	fbLys		: FB_Light_Type_A;
	
	stDaliSetup	: SH_Light.ST_DALI_RoomSetup := (		byShrtAdr_Prim := 10, 
														byGrpAdr_Prim := 2, 
														eMod_Prim := E_DALIAddressType.Group, 
													//	byShrtAdr_Sec := 1, 
													//	byGrpAdr_Sec := 1, 
													//	eMod_Sec := E_DALIAddressType.Short, 
													//	byShrtAdr_Supl := 1, 
														DALI_LINE_NUM_PRIM := 3, 
														DALI_LINE_NUM_SEC := 0, 
														DALI_LINE_NUM_SUPL := 0);
	stLiveData				: SH_Light.ST_LiveData;
	//stLiveData AT %MB22	: SH_Light.ST_LiveData;
	bTopButtonZone1			: BOOL;
	bTopButtonZone1_Visu	: BOOL;
	bBottomButtonZone1		: BOOL;
	bBottomButtonZone1_Visu	: BOOL;
	bButtonZone2			: BOOL;
	fLuxOn					: REAL;
	fLuxDim					: REAL;
	tPIRDim					: TIME;
	tPIROff					: TIME;
	fOffsetSec				: REAL := 20;
	bOccupiedRoom			: BOOL;

	bRunTuning				: BOOL;
	
// Sensor Settings
	//fbSensor					: SH_Light.FB_NIKO_P46xx_1Pcs;
	fbSensor					: SH_Light.FB_NIKO_P46xx_2Pcs;
	//bySensorAddr				: BYTE := 3;
	arrSensorAddr				: ARRAY[1..2] OF BYTE := [1,2];
	bInitialize					: BOOL := TRUE;
	stDaliSensorSetup			: ST_DALI_NIKOP46SetupData := (
																nSensitivityPIRSegmentA := arrSensitivityOccupancy[1],
																nSensitivityPIRSegmentB := arrSensitivityOccupancy[2],
																nSensitivityPIRSegmentC := arrSensitivityOccupancy[3]);
//	arrSensitivityOccupancy				: ARRAY[1..3] OF BYTE := [4,4,4];

	//bInitErr					: BOOL;
	//bInitDone					: BOOL;
	arrInitErr					: ARRAY [1..2] OF BOOL;
	arrInitDone					: ARRAY [1..2] OF BOOL;
	arrSensorScales				: ARRAY [1..10] OF SH_Light.ST_DALI_SensorScaleMode := [	(fMeassureMaxSensor := rMeassure_Zone5, fReadMaxSensor := rRead_Zone5),
																							(fMeassureMaxSensor := rMeassure_Zone5, fReadMaxSensor := rRead_Zone5),
																						8(())];
	bCancelHoldTimerOccupancy	: BOOL;
(*	eEventPriorityOccupancy		: E_DALIEventPriority := E_DALIEVENTPRIORITY.Middle;
	nHoldTimerOccupancy			: WORD := 5; // Value in s. 	
	nReportTimerOccupancy		: BYTE := 120; // Value in s, Preset manufacturer value
	nDeadtimeTimerOccupancy		: WORD := 100; // Value in ms, Predefined Value of DALI Standard
	bCancelHoldTimerOccupancy	: BOOL;
	nSensitivityOccupancy		: BYTE:= 3; //setting Sensivity (0..4) 0 (Off), 1 (Min), 2(Low), 3(High) and 4 (Max)

	bEnableLuxEvent				: BOOL;
	eEventPriorityBrightness	: E_DALIEventPriority := E_DALIEVENTPRIORITY.Middle;
	nDeadtimeTimerBrightness	: WORD := 1500; // Value in ms, Predefined Value of DALI Standard
	nHysteresisBrightness		: BYTE := 2; // Value in %
	nHysteresisMinBrightness	: BYTE := 10; // Absolute Value, depending on the manufacturer specific resolution
	nReportTimerBrightness		: BYTE := 120; // Value in s, Preset manufacturer value
*)



//ModbusComm setup
	
	fbWriteSPLuxLevel			: SH_Light.FB_TwoVal_SelectOne_RTrigChange;
	fbWritePirDelayTIme			: SH_Light.FB_TwoVal_SelectOne_RTrigChange;
	stRoomDataPLC				: SH_Light.ST_RoomDataPLC	:=	(	uiPirOffDelayTime	:= 30,
																	uiSpLuxLevel		:= 500,
																	uiPirDimDelayTime	:= 15,
																	uiSpDimLuxLevel		:= 200
																);
	fbBallastOnHours			: SH_Light.FB_CountOnHours;
	bEnableHourCount			: BOOL := TRUE;
	
	//Non-persistent modbus data
	bPirActive_MB			AT%MX32.0	: BOOL;				//bPirLys i gammel kode
	uiActLuxLevel_MB		AT%MB36	: UINT;				//intHMIAktueltLux i gammel kode
	uiActLightLevelPct_MB	AT%MB42		: UINT;				//intDALI_Gruppe1_Lysniveau i gammel kode
	
	//For Conversion
	uiPirOffMinutes						: UINT;
	udTimeScaling						: UDINT := 60000;
	uiLuxOn								: UINT;
	
	//max values checks
	uiMaxLuxLevel						: UINT := 1023;
	uiMaxPirOffMinutes					: UINT := 180;
	
END_VAR

VAR CONSTANT
Sensor_DALI_LINE_NUM: BYTE := 4;
	DALI_LINE_NUM_LIGHT: BYTE := 3;
	arrSensitivityOccupancy				: ARRAY[1..3] OF BYTE := [4,4,4];
END_VAR
VAR PERSISTENT
	stPirSensorData: SH_Light.ST_DALI_Sensor;
	stTuneData: SH_Light.ST_TuneData_EX;
	
	uiPirOffDelayTime_MB	AT%MB34		: UINT;				//ntHMI_Pir_SetValue i gammel kode
	uiSPLuxLevel_MB			AT%MB38 	: UINT;				//intHMI_Lux_SetValue i gammel kode
	uiBallastOnHours_MB		AT%MB46 	: UINT;				//dintHMILysbraendtimer1 i gammel kode
	byOnHoursOverflowCount				: BYTE;
END_VAR

A_Buttons();
A_LightCtrl();
A_Sensor();
A_Modbuscomm();

ACTION A_Buttons:
bTopButtonZone1		:= GVL_EnOcean.strEnOceanSwitch_Rum_3_329_Indgang.bT1_ON OR GVL_EnOcean.strEnOceanSwitch_Rum_3_329_Tavle.bT2_OFF OR bTopButtonZone1_Visu;
bBottomButtonZone1	:= GVL_EnOcean.strEnOceanSwitch_Rum_3_329_Indgang.bT1_OFF OR GVL_EnOcean.strEnOceanSwitch_Rum_3_329_Tavle.bT2_ON OR bBottomButtonZone1_Visu;
END_ACTION

ACTION A_LightCtrl:

fbLys(
	nZoneID:= 1, 
	bButtonZone1:= bTopButtonZone1,
	bBottomButtonZone1 := bBottomButtonZone1, 
	bButtonZone2:= bButtonZone2, 
	fLuxOn:= fLuxOn, 
	fLuxDim:= fLuxDim, 
	tPIRDim:= tPIRDim, 
	tPIROff:= tPIROff, 
	fOffsetSec:= fOffsetSec, 
	bReInit:= , 
	stDaliSetup:= stDaliSetup, 
	ipCommunication_Prim:= P_DALI_Background.arrfbKL6821Communication[DALI_LINE_NUM_LIGHT], 
//	ipCommunication_Sec:= P_DALI_Background.arrfbKL6821Communication[DALI_LINE_NUM_LIGHT], 
//	ipCommunication_Supl:= P_DALI_Background.arrfbKL6821Communication[DALI_LINE_NUM_LIGHT], 
	fMinOutputPowerLevelRoom:= 15, 
	fMaxOutputPowerLevelRoom:= 100, 
	nCycleTimeInMS:= SH_Light.DALI_Param.nPlcTaskCycleTimeInMS*nDimCmdCycleTimeFactor, 
	bRunTuning:= bRunTuning, 
	bOccupiedRoom=> bOccupiedRoom, 
	bError_Prim=> , 
	nError_Prim=> , 
	stTuneData:=stTuneData , 
	stPirSensorData:= stPirSensorData, 
	stLiveData:= stLiveData);
END_ACTION

ACTION A_ModbusComm:
//Manage data for modbus communication

//Manage data for read-only in PLC
stRoomDataPLC.bPirActive			:= stPirSensorData.bPrc;
stRoomDataPLC.uiActLuxLevel			:= TO_UINT(TRUNC(stPirSensorData.fBrightness));
stRoomDataPLC.uiActLightLevelPct	:= TO_UINT(TRUNC(fbLys.fbBallast.fActlLgtLvl_Prim));
		//stRoomDataPLC.uiActLightLevelPct	:= TO_UINT(TRUNC(fbLys.fbBallast.fActlLgtLvl_Prim)); //if only one group light control
stRoomDataPLC.uiBallastOnHours		:= uiBallastOnHours_MB; //The calculation for BallastOnHours is stored directly to the MB register below


//Assign data for read-only to MB registers
bPirActive_MB			:= stRoomDataPLC.bPirActive;
//uiActLuxLevel_MB		:= stRoomDataPLC.uiActLuxLevel;
uiActLightLevelPct_MB	:= stRoomDataPLC.uiActLightLevelPct;

	//calculate BallastOnHours
	fbBallastOnHours(
		bEnableHourCount	:= bEnableHourCount,
		bPauseCount			:= fbLys.fbLightCtrl.bOffZone1,
		uiOnHours			:= uiBallastOnHours_MB,			//OnHours is updated here
		byOverflowCount		:= byOnHoursOverflowCount);


//Manage data for read/write for both PLC and MB registers
fbWriteSPLuxLevel(	nMaxValOut	:= uiMaxLuxLevel,
					nValIn1		:= uiSPLuxLevel_MB,		//nValIn1 takes priotity in case of download or restart
					nValIn2		:= stRoomDataPLC.uiSpLuxLevel,
					nValOut		=> uiLuxOn
				);


fbWritePirDelayTIme(	nMaxValOut	:= uiMaxPirOffMinutes,
						nValIn1		:= uiPirOffDelayTime_MB,		//nValIn1 takes priotity in case of download or restart
						nValIn2		:= stRoomDataPLC.uiPirOffDelayTime,
						nValOut		=> uiPirOffMinutes
					);
					

//Convert read/write modbus data to appropriate datatypes in PLC
fLuxOn	:= TO_REAL(uiLuxOn);			
tPIROff	:= TO_TIME(uiPirOffMinutes*udTimeScaling); //Time conversion defaults to ms

fLuxDim	:= TO_REAL(stRoomDataPLC.uiSpDimLuxLevel);			
tPIRDim	:= TO_TIME(stRoomDataPLC.uiPirDimDelayTime*udTimeScaling); //Time conversion defaults to ms
END_ACTION

ACTION A_Sensor:

fbSensor.ipCommunication := P_DALI_Background.arrfbKL6821Communication[Sensor_DALI_LINE_NUM];

(*
fbSensor(
	byShrtAdr:= bySensorAddr,
	bInitialize:= bInitialize, 
	DALI_LINE_NUM:= Sensor_DALI_LINE_NUM, 
 	//bCancelHoldTimerOccupancy:= bCancelHoldTimerOccupancy, 
	stSensorSetup := stDaliSensorSetup,
	bInitErr=> bInitErr, 
	bInitDone=> bInitDone,
	stPirSensorData:= stPirSensorData, 
	arrSensorScales:= arrSensorScales);
	*)


fbSensor(
	arrShrtAdr:= arrSensorAddr,
	bInitialize:= bInitialize, 
	DALI_LINE_NUM:= Sensor_DALI_LINE_NUM, 
 	//bCancelHoldTimerOccupancy:= bCancelHoldTimerOccupancy, 
	stSensorSetup := stDaliSensorSetup,
	arrInitErr=> arrInitErr, 
	arrInitDone=> arrInitDone,
	stPirSensorData:= stPirSensorData, 
	arrSensorScales:= arrSensorScales);
END_ACTION

END_PROGRAM

// ---- POUs/Alle_Rum/Rum_Med_DALI_Pir/Rum_4_316/P_Rum_4_316.TcPOU
PROGRAM P_Rum_4_316
VAR
//Light

	fbLys		: FB_Light_Type_A;
	
	stDaliSetup	: SH_Light.ST_DALI_RoomSetup := (		byShrtAdr_Prim := 45, 
														byGrpAdr_Prim := 8, 
														eMod_Prim := E_DALIAddressType.Group, 
														//byShrtAdr_Sec := 1, 
														///byGrpAdr_Sec := 1, 
														//eMod_Sec := E_DALIAddressType.Short, 
														//byShrtAdr_Supl := 1, 
														DALI_LINE_NUM_PRIM := DALI_LINE_NUM_LIGHT, 
														DALI_LINE_NUM_SEC := 0, 
														DALI_LINE_NUM_SUPL := DALI_LINE_NUM_PENDANTS);
	stLiveData				: SH_Light.ST_LiveData;
	//stLiveData AT %MB22	: SH_Light.ST_LiveData;
	bTopButtonZone1			: BOOL;
	bTopButtonZone1_Visu	: BOOL;
	bBottomButtonZone1		: BOOL;
	bBottomButtonZone1_Visu	: BOOL;
	bButtonZone2			: BOOL;
	fLuxOn					: REAL;
	fLuxDim					: REAL;
	tPIRDim					: TIME;
	tPIROff					: TIME;
	fOffsetSec				: REAL := 20;
	bOccupiedRoom			: BOOL;

	bRunTuning				: BOOL;
	
// Sensor Settings
	fbSensor					: SH_Light.FB_NIKO_P46xx_1Pcs;
	//fbSensor					: SH_Light.FB_NIKO_P46xx_2Pcs;
	bySensorAddr				: BYTE := 4;
	//arrSensorAddr				: ARRAY[1..2] OF BYTE := [9,10];
	bInitialize					: BOOL := TRUE;
	stDaliSensorSetup			: ST_DALI_NIKOP46SetupData := (
																nSensitivityPIRSegmentA := arrSensitivityOccupancy[1],
																nSensitivityPIRSegmentB := arrSensitivityOccupancy[2],
																nSensitivityPIRSegmentC := arrSensitivityOccupancy[3]);
//	arrSensitivityOccupancy				: ARRAY[1..3] OF BYTE := [4,4,4];
	bInitErr					: BOOL;
	bInitDone					: BOOL;
	//arrInitErr					: ARRAY [1..2] OF BOOL;
	//arrInitDone					: ARRAY [1..2] OF BOOL;
	arrSensorScales				: ARRAY [1..10] OF SH_Light.ST_DALI_SensorScaleMode := [	(fMeassureMaxSensor := rMeassure_Zone10, fReadMaxSensor := rRead_Zone10),
																						9(())];
	bCancelHoldTimerOccupancy	: BOOL;
(*	eEventPriorityOccupancy		: E_DALIEventPriority := E_DALIEVENTPRIORITY.Middle;
	nHoldTimerOccupancy			: WORD := 5; // Value in s. 	
	nReportTimerOccupancy		: BYTE := 120; // Value in s, Preset manufacturer value
	nDeadtimeTimerOccupancy		: WORD := 100; // Value in ms, Predefined Value of DALI Standard
	bCancelHoldTimerOccupancy	: BOOL;
	nSensitivityOccupancy		: BYTE:= 3; //setting Sensivity (0..4) 0 (Off), 1 (Min), 2(Low), 3(High) and 4 (Max)

	bEnableLuxEvent				: BOOL;
	eEventPriorityBrightness	: E_DALIEventPriority := E_DALIEVENTPRIORITY.Middle;
	nDeadtimeTimerBrightness	: WORD := 1500; // Value in ms, Predefined Value of DALI Standard
	nHysteresisBrightness		: BYTE := 2; // Value in %
	nHysteresisMinBrightness	: BYTE := 10; // Absolute Value, depending on the manufacturer specific resolution
	nReportTimerBrightness		: BYTE := 120; // Value in s, Preset manufacturer value
*)



//ModbusComm setup
	
	fbWriteSPLuxLevel			: SH_Light.FB_TwoVal_SelectOne_RTrigChange;
	fbWritePirDelayTIme			: SH_Light.FB_TwoVal_SelectOne_RTrigChange;
	stRoomDataPLC				: SH_Light.ST_RoomDataPLC	:=	(	uiPirOffDelayTime	:= 30,
																	uiSpLuxLevel		:= 500,
																	uiPirDimDelayTime	:= 15,
																	uiSpDimLuxLevel		:= 200
																);
	fbBallastOnHours			: SH_Light.FB_CountOnHours;
	bEnableHourCount			: BOOL := TRUE;
	
	//Non-persistent modbus data
	bPirActive_MB			AT%MX172.0	    : BOOL;				//bPirLys i gammel kode
	uiActLuxLevel_MB		AT%MB300		         : UINT;				//intHMIAktueltLux i gammel kode
	uiActLightLevelPct_MB	AT%MB176		: UINT;				//intDALI_Gruppe1_Lysniveau i gammel kode
	
	//For Conversion
	uiPirOffMinutes						: UINT;
	udTimeScaling						: UDINT := 60000;
	uiLuxOn								: UINT;
	
	//max values checks
	uiMaxLuxLevel						: UINT := 1023;
	uiMaxPirOffMinutes					: UINT := 180;
	
END_VAR

VAR CONSTANT
	Sensor_DALI_LINE_NUM	: BYTE := 2;
	DALI_LINE_NUM_LIGHT		: BYTE := 1;
	DALI_LINE_NUM_PENDANTS	: BYTE := 0;
	arrSensitivityOccupancy				: ARRAY[1..3] OF BYTE := [4,4,4];
END_VAR
VAR PERSISTENT
	stPirSensorData: SH_Light.ST_DALI_Sensor;
	stTuneData: SH_Light.ST_TuneData_EX;
	
	uiPirOffDelayTime_MB	AT%MB174	: UINT;				//ntHMI_Pir_SetValue i gammel kode
	uiSPLuxLevel_MB			AT%MB302	     	: UINT;				//intHMI_Lux_SetValue i gammel kode
	uiBallastOnHours_MB		AT%MB178	: UINT;				//dintHMILysbraendtimer1 i gammel kode
	byOnHoursOverflowCount				: BYTE;
END_VAR

A_Buttons();
A_LightCtrl();
A_Sensor();
A_ModbusComm();

ACTION A_Buttons:
bTopButtonZone1		:= GVL_EnOcean.strEnOceanSwitch_Rum_4_316.bT2_ON OR bTopButtonZone1_Visu;
bBottomButtonZone1	:= GVL_EnOcean.strEnOceanSwitch_Rum_4_316.bT2_OFF OR bBottomButtonZone1_Visu;
END_ACTION

ACTION A_LightCtrl:

fbLys(
	nZoneID:= 1, 
	bButtonZone1:= bTopButtonZone1,
	bBottomButtonZone1 := bBottomButtonZone1, 
	bButtonZone2:= bButtonZone2, 
	fLuxOn:= fLuxOn, 
	fLuxDim:= fLuxDim, 
	tPIRDim:= tPIRDim, 
	tPIROff:= tPIROff, 
	fOffsetSec:= fOffsetSec, 
	bReInit:= , 
	stDaliSetup:= stDaliSetup, 
	ipCommunication_Prim:= P_DALI_Background.arrfbKL6821Communication[DALI_LINE_NUM_LIGHT], 
//	ipCommunication_Sec:= P_DALI_Background.arrfbKL6821Communication[DALI_LINE_NUM_LIGHT], 
//	ipCommunication_Supl:= P_DALI_Background.arrfbKL6821Communication[DALI_LINE_NUM_LIGHT], 
	fMinOutputPowerLevelRoom:= 15, 
	fMaxOutputPowerLevelRoom:= 100, 
	nCycleTimeInMS:= SH_Light.DALI_Param.nPlcTaskCycleTimeInMS*nDimCmdCycleTimeFactor , 
	bRunTuning:= bRunTuning, 
	bOccupiedRoom=> bOccupiedRoom, 
	bError_Prim=> , 
	nError_Prim=> , 
	stTuneData:=stTuneData , 
	stPirSensorData:= stPirSensorData, 
	stLiveData:= stLiveData);
END_ACTION

ACTION A_ModbusComm:
//Manage data for modbus communication

//Manage data for read-only in PLC
stRoomDataPLC.bPirActive			:= stPirSensorData.bPrc;
stRoomDataPLC.uiActLuxLevel			:= TO_UINT(TRUNC(stPirSensorData.fBrightness));
stRoomDataPLC.uiActLightLevelPct	:= TO_UINT(TRUNC(fbLys.fbBallast.fActlLgtLvl_Prim));
		//stRoomDataPLC.uiActLightLevelPct	:= TO_UINT(TRUNC(fbLys.fbBallast.fActlLgtLvl_Prim)); //if only one group light control
stRoomDataPLC.uiBallastOnHours		:= uiBallastOnHours_MB; //The calculation for BallastOnHours is stored directly to the MB register below


//Assign data for read-only to MB registers
bPirActive_MB			:= stRoomDataPLC.bPirActive;
//uiActLuxLevel_MB		:= stRoomDataPLC.uiActLuxLevel;
uiActLightLevelPct_MB	:= stRoomDataPLC.uiActLightLevelPct;

	//calculate BallastOnHours
	fbBallastOnHours(
		bEnableHourCount	:= bEnableHourCount,
		bPauseCount			:= fbLys.fbLightCtrl.bOffZone1,
		uiOnHours			:= uiBallastOnHours_MB,			//OnHours is updated here
		byOverflowCount		:= byOnHoursOverflowCount);


//Manage data for read/write for both PLC and MB registers
fbWriteSPLuxLevel(	nMaxValOut	:= uiMaxLuxLevel,
					nValIn1		:= uiSPLuxLevel_MB,		//nValIn1 takes priotity in case of download or restart
					nValIn2		:= stRoomDataPLC.uiSpLuxLevel,
					nValOut		=> uiLuxOn
				);


fbWritePirDelayTIme(	nMaxValOut	:= uiMaxPirOffMinutes,
						nValIn1		:= uiPirOffDelayTime_MB,		//nValIn1 takes priotity in case of download or restart
						nValIn2		:= stRoomDataPLC.uiPirOffDelayTime,
						nValOut		=> uiPirOffMinutes
					);
					

//Convert read/write modbus data to appropriate datatypes in PLC
fLuxOn	:= TO_REAL(uiLuxOn);			
tPIROff	:= TO_TIME(uiPirOffMinutes*udTimeScaling); //Time conversion defaults to ms

fLuxDim	:= TO_REAL(stRoomDataPLC.uiSpDimLuxLevel);			
tPIRDim	:= TO_TIME(stRoomDataPLC.uiPirDimDelayTime*udTimeScaling); //Time conversion defaults to ms
END_ACTION

ACTION A_Sensor:

fbSensor.ipCommunication := P_DALI_Background.arrfbKL6821Communication[Sensor_DALI_LINE_NUM];


fbSensor(
	byShrtAdr:= bySensorAddr,
	bInitialize:= bInitialize, 
	DALI_LINE_NUM:= Sensor_DALI_LINE_NUM, 
 	//bCancelHoldTimerOccupancy:= bCancelHoldTimerOccupancy, 
	stSensorSetup := stDaliSensorSetup,
	bInitErr=> bInitErr, 
	bInitDone=> bInitDone,
	stPirSensorData:= stPirSensorData, 
	arrSensorScales:= arrSensorScales);

(*
fbSensor(
	arrShrtAdr:= arrSensorAddr,
	bInitialize:= bInitialize, 
	DALI_LINE_NUM:= Sensor_DALI_LINE_NUM, 
 	//bCancelHoldTimerOccupancy:= bCancelHoldTimerOccupancy, 
	stSensorSetup := stDaliSensorSetup,
	arrInitErr=> arrInitErr, 
	arrInitDone=> arrInitDone,
	stPirSensorData:= stPirSensorData, 
	arrSensorScales:= arrSensorScales);
	*)
END_ACTION

END_PROGRAM

// ---- POUs/Alle_Rum/Rum_Med_DALI_Pir/Rum_4_321/P_Rum_4_321.TcPOU
PROGRAM P_Rum_4_321
VAR
//Light

	fbLys		: FB_Light_Type_A;
	
	stDaliSetup	: SH_Light.ST_DALI_RoomSetup := (		byShrtAdr_Prim := 37, 
														byGrpAdr_Prim := 7, 
														eMod_Prim := E_DALIAddressType.Group, 
												//		byShrtAdr_Sec := 1, 
												//		byGrpAdr_Sec := 1, 
												//		eMod_Sec := E_DALIAddressType.Short, 
												//		byShrtAdr_Supl := 1, 
														DALI_LINE_NUM_PRIM := DALI_LINE_NUM_LIGHT, 
														DALI_LINE_NUM_SEC := 0, 
														DALI_LINE_NUM_SUPL := DALI_LINE_NUM_PENDANTS);
	stLiveData				: SH_Light.ST_LiveData;
	//stLiveData AT %MB22	: SH_Light.ST_LiveData;
	bTopButtonZone1			: BOOL;
	bTopButtonZone1_Visu	: BOOL;
	bBottomButtonZone1		: BOOL;
	bBottomButtonZone1_Visu	: BOOL;
	bButtonZone2			: BOOL;
	fLuxOn					: REAL;
	fLuxDim					: REAL;
	tPIRDim					: TIME;
	tPIROff					: TIME;
	fOffsetSec				: REAL := 20;
	bOccupiedRoom			: BOOL;

	bRunTuning				: BOOL;
	
// Sensor Settings
	fbSensor					: SH_Light.FB_NIKO_P46xx_1Pcs;
	//fbSensor					: SH_Light.FB_NIKO_P46xx_2Pcs;
	bySensorAddr				: BYTE := 3;
	//arrSensorAddr				: ARRAY[1..2] OF BYTE := [9,10];
	bInitialize					: BOOL := TRUE;
	stDaliSensorSetup			: ST_DALI_NIKOP46SetupData := (
																nSensitivityPIRSegmentA := arrSensitivityOccupancy[1],
																nSensitivityPIRSegmentB := arrSensitivityOccupancy[2],
																nSensitivityPIRSegmentC := arrSensitivityOccupancy[3]);
//	arrSensitivityOccupancy				: ARRAY[1..3] OF BYTE := [4,4,4];
	bInitErr					: BOOL;
	bInitDone					: BOOL;
	//arrInitErr					: ARRAY [1..2] OF BOOL;
	//arrInitDone					: ARRAY [1..2] OF BOOL;
	arrSensorScales				: ARRAY [1..10] OF SH_Light.ST_DALI_SensorScaleMode := [	(fMeassureMaxSensor := rMeassure_Zone5, fReadMaxSensor := rRead_Zone5),
																						9(())];
	bCancelHoldTimerOccupancy	: BOOL;
(*	eEventPriorityOccupancy		: E_DALIEventPriority := E_DALIEVENTPRIORITY.Middle;
	nHoldTimerOccupancy			: WORD := 5; // Value in s. 	
	nReportTimerOccupancy		: BYTE := 120; // Value in s, Preset manufacturer value
	nDeadtimeTimerOccupancy		: WORD := 100; // Value in ms, Predefined Value of DALI Standard
	bCancelHoldTimerOccupancy	: BOOL;
	nSensitivityOccupancy		: BYTE:= 3; //setting Sensivity (0..4) 0 (Off), 1 (Min), 2(Low), 3(High) and 4 (Max)

	bEnableLuxEvent				: BOOL;
	eEventPriorityBrightness	: E_DALIEventPriority := E_DALIEVENTPRIORITY.Middle;
	nDeadtimeTimerBrightness	: WORD := 1500; // Value in ms, Predefined Value of DALI Standard
	nHysteresisBrightness		: BYTE := 2; // Value in %
	nHysteresisMinBrightness	: BYTE := 10; // Absolute Value, depending on the manufacturer specific resolution
	nReportTimerBrightness		: BYTE := 120; // Value in s, Preset manufacturer value
*)




//ModbusComm setup
	
	fbWriteSPLuxLevel			: SH_Light.FB_TwoVal_SelectOne_RTrigChange;
	fbWritePirDelayTIme			: SH_Light.FB_TwoVal_SelectOne_RTrigChange;
	stRoomDataPLC				: SH_Light.ST_RoomDataPLC	:=	(	uiPirOffDelayTime	:= 30,
																	uiSpLuxLevel		:= 500,
																	uiPirDimDelayTime	:= 15,
																	uiSpDimLuxLevel		:= 200
																);
	fbBallastOnHours			: SH_Light.FB_CountOnHours;
	bEnableHourCount			: BOOL := TRUE;
	
	//Non-persistent modbus data
	bPirActive_MB			AT%MX180.0	: BOOL;				//bPirLys i gammel kode
	uiActLuxLevel_MB		AT%MB184	: UINT;				//intHMIAktueltLux i gammel kode
	uiActLightLevelPct_MB	AT%MB188		: UINT;				//intDALI_Gruppe1_Lysniveau i gammel kode
	
	//For Conversion
	uiPirOffMinutes						: UINT;
	udTimeScaling						: UDINT := 60000;
	uiLuxOn								: UINT;
	
	//max values checks
	uiMaxLuxLevel						: UINT := 1023;
	uiMaxPirOffMinutes					: UINT := 180;
	
END_VAR

VAR CONSTANT
	Sensor_DALI_LINE_NUM	: BYTE := 2;
	DALI_LINE_NUM_LIGHT		: BYTE := 1;
	DALI_LINE_NUM_PENDANTS	: BYTE := 0;
	arrSensitivityOccupancy				: ARRAY[1..3] OF BYTE := [4,4,4];
END_VAR
VAR PERSISTENT
	stPirSensorData: SH_Light.ST_DALI_Sensor;
	stTuneData: SH_Light.ST_TuneData_EX;
	
	uiPirOffDelayTime_MB	AT%MB182	: UINT;				//ntHMI_Pir_SetValue i gammel kode
	uiSPLuxLevel_MB			AT%MB186 	: UINT;				//intHMI_Lux_SetValue i gammel kode
	uiBallastOnHours_MB		AT%MB190	: UINT;				//dintHMILysbraendtimer1 i gammel kode
	byOnHoursOverflowCount				: BYTE;
END_VAR

A_Buttons();
A_LightCtrl();
A_Sensor();
A_Modbuscomm();

ACTION A_Buttons:
bTopButtonZone1		:= GVL_EnOcean.strEnOceanSwitch_Rum_4_321.bT2_ON OR bTopButtonZone1_Visu;
bBottomButtonZone1	:= GVL_EnOcean.strEnOceanSwitch_Rum_4_321.bT2_OFF OR bBottomButtonZone1_Visu;
END_ACTION

ACTION A_LightCtrl:

fbLys(
	nZoneID:= 1, 
	bButtonZone1:= bTopButtonZone1,
	bBottomButtonZone1 := bBottomButtonZone1, 
	bButtonZone2:= bButtonZone2, 
	fLuxOn:= fLuxOn, 
	fLuxDim:= fLuxDim, 
	tPIRDim:= tPIRDim, 
	tPIROff:= tPIROff, 
	fOffsetSec:= fOffsetSec, 
	bReInit:= , 
	stDaliSetup:= stDaliSetup, 
	ipCommunication_Prim:= P_DALI_Background.arrfbKL6821Communication[DALI_LINE_NUM_LIGHT], 
//	ipCommunication_Sec:= P_DALI_Background.arrfbKL6821Communication[DALI_LINE_NUM_LIGHT], 
//	ipCommunication_Supl:= P_DALI_Background.arrfbKL6821Communication[DALI_LINE_NUM_LIGHT], 
	fMinOutputPowerLevelRoom:= 15, 
	fMaxOutputPowerLevelRoom:= 100, 
	nCycleTimeInMS:= SH_Light.DALI_Param.nPlcTaskCycleTimeInMS*nDimCmdCycleTimeFactor, 
	bRunTuning:= bRunTuning, 
	bOccupiedRoom=> bOccupiedRoom, 
	bError_Prim=> , 
	nError_Prim=> , 
	stTuneData:=stTuneData , 
	stPirSensorData:= stPirSensorData, 
	stLiveData:= stLiveData);
END_ACTION

ACTION A_ModbusComm:
//Manage data for modbus communication

//Manage data for read-only in PLC
stRoomDataPLC.bPirActive			:= stPirSensorData.bPrc;
stRoomDataPLC.uiActLuxLevel			:= TO_UINT(TRUNC(stPirSensorData.fBrightness));
stRoomDataPLC.uiActLightLevelPct	:= TO_UINT(TRUNC(fbLys.fbBallast.fActlLgtLvl_Prim));
		//stRoomDataPLC.uiActLightLevelPct	:= TO_UINT(TRUNC(fbLys.fbBallast.fActlLgtLvl_Prim)); //if only one group light control
stRoomDataPLC.uiBallastOnHours		:= uiBallastOnHours_MB; //The calculation for BallastOnHours is stored directly to the MB register below


//Assign data for read-only to MB registers
bPirActive_MB			:= stRoomDataPLC.bPirActive;
//uiActLuxLevel_MB		:= stRoomDataPLC.uiActLuxLevel;
uiActLightLevelPct_MB	:= stRoomDataPLC.uiActLightLevelPct;

	//calculate BallastOnHours
	fbBallastOnHours(
		bEnableHourCount	:= bEnableHourCount,
		bPauseCount			:= fbLys.fbLightCtrl.bOffZone1,
		uiOnHours			:= uiBallastOnHours_MB,			//OnHours is updated here
		byOverflowCount		:= byOnHoursOverflowCount);


//Manage data for read/write for both PLC and MB registers
fbWriteSPLuxLevel(	nMaxValOut	:= uiMaxLuxLevel,
					nValIn1		:= uiSPLuxLevel_MB,		//nValIn1 takes priotity in case of download or restart
					nValIn2		:= stRoomDataPLC.uiSpLuxLevel,
					nValOut		=> uiLuxOn
				);


fbWritePirDelayTIme(	nMaxValOut	:= uiMaxPirOffMinutes,
						nValIn1		:= uiPirOffDelayTime_MB,		//nValIn1 takes priotity in case of download or restart
						nValIn2		:= stRoomDataPLC.uiPirOffDelayTime,
						nValOut		=> uiPirOffMinutes
					);
					

//Convert read/write modbus data to appropriate datatypes in PLC
fLuxOn	:= TO_REAL(uiLuxOn);			
tPIROff	:= TO_TIME(uiPirOffMinutes*udTimeScaling); //Time conversion defaults to ms

fLuxDim	:= TO_REAL(stRoomDataPLC.uiSpDimLuxLevel);			
tPIRDim	:= TO_TIME(stRoomDataPLC.uiPirDimDelayTime*udTimeScaling); //Time conversion defaults to ms
END_ACTION

ACTION A_Sensor:

fbSensor.ipCommunication := P_DALI_Background.arrfbKL6821Communication[Sensor_DALI_LINE_NUM];


fbSensor(
	byShrtAdr:= bySensorAddr,
	bInitialize:= bInitialize, 
	DALI_LINE_NUM:= Sensor_DALI_LINE_NUM, 
 	//bCancelHoldTimerOccupancy:= bCancelHoldTimerOccupancy, 
	stSensorSetup := stDaliSensorSetup,
	bInitErr=> bInitErr, 
	bInitDone=> bInitDone,
	stPirSensorData:= stPirSensorData, 
	arrSensorScales:= arrSensorScales);

(*
fbSensor(
	arrShrtAdr:= arrSensorAddr,
	bInitialize:= bInitialize, 
	DALI_LINE_NUM:= Sensor_DALI_LINE_NUM, 
 	//bCancelHoldTimerOccupancy:= bCancelHoldTimerOccupancy, 
	stSensorSetup := stDaliSensorSetup,
	arrInitErr=> arrInitErr, 
	arrInitDone=> arrInitDone,
	stPirSensorData:= stPirSensorData, 
	arrSensorScales:= arrSensorScales);
	*)
END_ACTION

END_PROGRAM

// ---- POUs/Alle_Rum/Rum_Med_DALI_Pir/Rum_4_322/P_Rum_4_322.TcPOU
PROGRAM P_Rum_4_322
VAR
//Light

	fbLys		: FB_Light_Type_A;
	
	stDaliSetup	: SH_Light.ST_DALI_RoomSetup := (		byShrtAdr_Prim := 49, 
														byGrpAdr_Prim := 9, 
														eMod_Prim := E_DALIAddressType.Group, 
														//byShrtAdr_Sec := 1, 
														//byGrpAdr_Sec := 1, 
														//eMod_Sec := E_DALIAddressType.Short, 
														//byShrtAdr_Supl := 1, 
														DALI_LINE_NUM_PRIM := DALI_LINE_NUM_LIGHT, 
														DALI_LINE_NUM_SEC := 0, 
														DALI_LINE_NUM_SUPL := DALI_LINE_NUM_PENDANTS);
	stLiveData				: SH_Light.ST_LiveData;
	//stLiveData AT %MB22	: SH_Light.ST_LiveData;
	bTopButtonZone1			: BOOL;
	bTopButtonZone1_Visu	: BOOL;
	bBottomButtonZone1		: BOOL;
	bBottomButtonZone1_Visu	: BOOL;
	bButtonZone2			: BOOL;
	fLuxOn					: REAL;
	fLuxDim					: REAL;
	tPIRDim					: TIME;
	tPIROff					: TIME;
	fOffsetSec				: REAL := 20;
	bOccupiedRoom			: BOOL;

	bRunTuning				: BOOL;
	
// Sensor Settings
	fbSensor					: SH_Light.FB_NIKO_P46xx_1Pcs;
	//fbSensor					: SH_Light.FB_NIKO_P46xx_2Pcs;
	bySensorAddr				: BYTE := 5;
	//arrSensorAddr				: ARRAY[1..2] OF BYTE := [9,10];
	bInitialize					: BOOL := TRUE;
	stDaliSensorSetup			: ST_DALI_NIKOP46SetupData := (
																nSensitivityPIRSegmentA := arrSensitivityOccupancy[1],
																nSensitivityPIRSegmentB := arrSensitivityOccupancy[2],
																nSensitivityPIRSegmentC := arrSensitivityOccupancy[3]);
//	arrSensitivityOccupancy				: ARRAY[1..3] OF BYTE := [4,4,4];
	bInitErr					: BOOL;
	bInitDone					: BOOL;
	//arrInitErr					: ARRAY [1..2] OF BOOL;
	//arrInitDone					: ARRAY [1..2] OF BOOL;
	arrSensorScales				: ARRAY [1..10] OF SH_Light.ST_DALI_SensorScaleMode := [	(fMeassureMaxSensor := rMeassure_Zone10, fReadMaxSensor := rRead_Zone10),
																						9(())];
	bCancelHoldTimerOccupancy	: BOOL;
(*	eEventPriorityOccupancy		: E_DALIEventPriority := E_DALIEVENTPRIORITY.Middle;
	nHoldTimerOccupancy			: WORD := 5; // Value in s. 	
	nReportTimerOccupancy		: BYTE := 120; // Value in s, Preset manufacturer value
	nDeadtimeTimerOccupancy		: WORD := 100; // Value in ms, Predefined Value of DALI Standard
	bCancelHoldTimerOccupancy	: BOOL;
	nSensitivityOccupancy		: BYTE:= 3; //setting Sensivity (0..4) 0 (Off), 1 (Min), 2(Low), 3(High) and 4 (Max)

	bEnableLuxEvent				: BOOL;
	eEventPriorityBrightness	: E_DALIEventPriority := E_DALIEVENTPRIORITY.Middle;
	nDeadtimeTimerBrightness	: WORD := 1500; // Value in ms, Predefined Value of DALI Standard
	nHysteresisBrightness		: BYTE := 2; // Value in %
	nHysteresisMinBrightness	: BYTE := 10; // Absolute Value, depending on the manufacturer specific resolution
	nReportTimerBrightness		: BYTE := 120; // Value in s, Preset manufacturer value
*)



//ModbusComm setup
	
	fbWriteSPLuxLevel			: SH_Light.FB_TwoVal_SelectOne_RTrigChange;
	fbWritePirDelayTIme			: SH_Light.FB_TwoVal_SelectOne_RTrigChange;
	stRoomDataPLC				: SH_Light.ST_RoomDataPLC	:=	(	uiPirOffDelayTime	:= 30,
																	uiSpLuxLevel		:= 500,
																	uiPirDimDelayTime	:= 15,
																	uiSpDimLuxLevel		:= 200
																);
	fbBallastOnHours			: SH_Light.FB_CountOnHours;
	bEnableHourCount			: BOOL := TRUE;
	
	//Non-persistent modbus data
	bPirActive_MB			AT%MX196.0	: BOOL;				//bPirLys i gammel kode
	uiActLuxLevel_MB		AT%MB304		: UINT;				//intHMIAktueltLux i gammel kode
	uiActLightLevelPct_MB	AT%MB200		: UINT;				//intDALI_Gruppe1_Lysniveau i gammel kode
	
	//For Conversion
	uiPirOffMinutes						: UINT;
	udTimeScaling						: UDINT := 60000;
	uiLuxOn								: UINT;
	
	//max values checks
	uiMaxLuxLevel						: UINT := 1023;
	uiMaxPirOffMinutes					: UINT := 180;
	
END_VAR

VAR CONSTANT
	Sensor_DALI_LINE_NUM	: BYTE := 2;
	DALI_LINE_NUM_LIGHT		: BYTE := 1;
	DALI_LINE_NUM_PENDANTS	: BYTE := 0;
	arrSensitivityOccupancy				: ARRAY[1..3] OF BYTE := [4,4,4];
END_VAR
VAR PERSISTENT
	stPirSensorData: SH_Light.ST_DALI_Sensor;
	stTuneData: SH_Light.ST_TuneData_EX;
	
	uiPirOffDelayTime_MB	AT%MB198	: UINT;				//tHMI_Pir_SetValue i gammel koden
	uiSPLuxLevel_MB			AT%MB306 	: UINT;				//intHMI_Lux_SetValue i gammel kode
	uiBallastOnHours_MB		AT%MB202	: UINT;				//dintHMILysbraendtimer1 i gammel kode
	byOnHoursOverflowCount				: BYTE;
END_VAR

A_Buttons();
A_LightCtrl();
A_Sensor();
A_ModbusComm();

ACTION A_Buttons:
bTopButtonZone1		:= GVL_EnOcean.strEnOceanSwitch_Rum_4_322.bT2_ON OR bTopButtonZone1_Visu;
bBottomButtonZone1	:= GVL_EnOcean.strEnOceanSwitch_Rum_4_322.bT2_OFF OR bBottomButtonZone1_Visu;
END_ACTION

ACTION A_LightCtrl:

fbLys(
	nZoneID:= 1, 
	bButtonZone1:= bTopButtonZone1,
	bBottomButtonZone1 := bBottomButtonZone1, 
	bButtonZone2:= bButtonZone2, 
	fLuxOn:= fLuxOn, 
	fLuxDim:= fLuxDim, 
	tPIRDim:= tPIRDim, 
	tPIROff:= tPIROff, 
	fOffsetSec:= fOffsetSec, 
	bReInit:= , 
	stDaliSetup:= stDaliSetup, 
	ipCommunication_Prim:= P_DALI_Background.arrfbKL6821Communication[DALI_LINE_NUM_LIGHT], 
//	ipCommunication_Sec:= P_DALI_Background.arrfbKL6821Communication[DALI_LINE_NUM_LIGHT], 
//	ipCommunication_Supl:= P_DALI_Background.arrfbKL6821Communication[DALI_LINE_NUM_LIGHT], 
	fMinOutputPowerLevelRoom:= 15, 
	fMaxOutputPowerLevelRoom:= 100, 
	nCycleTimeInMS:= SH_Light.DALI_Param.nPlcTaskCycleTimeInMS*nDimCmdCycleTimeFactor, 
	bRunTuning:= bRunTuning, 
	bOccupiedRoom=> bOccupiedRoom, 
	bError_Prim=> , 
	nError_Prim=> , 
	stTuneData:=stTuneData , 
	stPirSensorData:= stPirSensorData, 
	stLiveData:= stLiveData);
END_ACTION

ACTION A_ModbusComm:
//Manage data for modbus communication

//Manage data for read-only in PLC
stRoomDataPLC.bPirActive			:= stPirSensorData.bPrc;
stRoomDataPLC.uiActLuxLevel			:= TO_UINT(TRUNC(stPirSensorData.fBrightness));
stRoomDataPLC.uiActLightLevelPct	:= TO_UINT(TRUNC(fbLys.fbBallast.fActlLgtLvl_Prim));
		//stRoomDataPLC.uiActLightLevelPct	:= TO_UINT(TRUNC(fbLys.fbBallast.fActlLgtLvl_Prim)); //if only one group light control
stRoomDataPLC.uiBallastOnHours		:= uiBallastOnHours_MB; //The calculation for BallastOnHours is stored directly to the MB register below


//Assign data for read-only to MB registers
bPirActive_MB			:= stRoomDataPLC.bPirActive;
//uiActLuxLevel_MB		:= stRoomDataPLC.uiActLuxLevel;
uiActLightLevelPct_MB	:= stRoomDataPLC.uiActLightLevelPct;

	//calculate BallastOnHours
	fbBallastOnHours(
		bEnableHourCount	:= bEnableHourCount,
		bPauseCount			:= fbLys.fbLightCtrl.bOffZone1,
		uiOnHours			:= uiBallastOnHours_MB,			//OnHours is updated here
		byOverflowCount		:= byOnHoursOverflowCount);


//Manage data for read/write for both PLC and MB registers
fbWriteSPLuxLevel(	nMaxValOut	:= uiMaxLuxLevel,
					nValIn1		:= uiSPLuxLevel_MB,		//nValIn1 takes priotity in case of download or restart
					nValIn2		:= stRoomDataPLC.uiSpLuxLevel,
					nValOut		=> uiLuxOn
				);


fbWritePirDelayTIme(	nMaxValOut	:= uiMaxPirOffMinutes,
						nValIn1		:= uiPirOffDelayTime_MB,		//nValIn1 takes priotity in case of download or restart
						nValIn2		:= stRoomDataPLC.uiPirOffDelayTime,
						nValOut		=> uiPirOffMinutes
					);
					

//Convert read/write modbus data to appropriate datatypes in PLC
fLuxOn	:= TO_REAL(uiLuxOn);			
tPIROff	:= TO_TIME(uiPirOffMinutes*udTimeScaling); //Time conversion defaults to ms

fLuxDim	:= TO_REAL(stRoomDataPLC.uiSpDimLuxLevel);			
tPIRDim	:= TO_TIME(stRoomDataPLC.uiPirDimDelayTime*udTimeScaling); //Time conversion defaults to ms
END_ACTION

ACTION A_Sensor:

fbSensor.ipCommunication := P_DALI_Background.arrfbKL6821Communication[Sensor_DALI_LINE_NUM];


fbSensor(
	byShrtAdr:= bySensorAddr,
	bInitialize:= bInitialize, 
	DALI_LINE_NUM:= Sensor_DALI_LINE_NUM, 
 	//bCancelHoldTimerOccupancy:= bCancelHoldTimerOccupancy, 
	stSensorSetup := stDaliSensorSetup,
	bInitErr=> bInitErr, 
	bInitDone=> bInitDone,
	stPirSensorData:= stPirSensorData, 
	arrSensorScales:= arrSensorScales);

(*
fbSensor(
	arrShrtAdr:= arrSensorAddr,
	bInitialize:= bInitialize, 
	DALI_LINE_NUM:= Sensor_DALI_LINE_NUM, 
 	//bCancelHoldTimerOccupancy:= bCancelHoldTimerOccupancy, 
	stSensorSetup := stDaliSensorSetup,
	arrInitErr=> arrInitErr, 
	arrInitDone=> arrInitDone,
	stPirSensorData:= stPirSensorData, 
	arrSensorScales:= arrSensorScales);
	*)
END_ACTION

END_PROGRAM

// ---- POUs/Alle_Rum/Rum_Med_DALI_Pir/Rum_4_325_template/P_Rum_4_325.TcPOU
PROGRAM P_Rum_4_325
VAR
//Light

	fbLys		: FB_Light_Type_A;
	
	stDaliSetup	: SH_Light.ST_DALI_RoomSetup := (		byShrtAdr_Prim := 1, 
														byGrpAdr_Prim := 1, 
														eMod_Prim := E_DALIAddressType.Group, 
														byShrtAdr_Sec := 1, 
														byGrpAdr_Sec := 1, 
														eMod_Sec := E_DALIAddressType.Short, 
														byShrtAdr_Supl := 1, 
														DALI_LINE_NUM_PRIM := DALI_LINE_NUM_LIGHT, 
														DALI_LINE_NUM_SEC := 0, //0 = ingen zonestyring/vinduerække
														DALI_LINE_NUM_SUPL := DALI_LINE_NUM_PENDANTS);
	stLiveData				: SH_Light.ST_LiveData;
	//stLiveData AT %MB22	: SH_Light.ST_LiveData;
	bTopButtonZone1			: BOOL;
	bTopButtonZone1_Visu	: BOOL;
	bBottomButtonZone1		: BOOL;
	bBottomButtonZone1_Visu	: BOOL;
	bButtonZone2			: BOOL;
	fLuxOn					: REAL;
	fLuxDim					: REAL;
	tPIRDim					: TIME;
	tPIROff					: TIME;
	fOffsetSec				: REAL := 20;
	bOccupiedRoom			: BOOL;

	bRunTuning				: BOOL;
	
// Sensor Settings
	fbSensor					: SH_Light.FB_NIKO_P46xx_1Pcs;
	//fbSensor					: SH_Light.FB_NIKO_P46xx_2Pcs;
	bySensorAddr				: BYTE := 1;
	//arrSensorAddr				: ARRAY[1..2] OF BYTE := [9,10];
	bInitialize					: BOOL := TRUE;
	stDaliSensorSetup			: ST_DALI_NIKOP46SetupData;
	bInitErr					: BOOL;
	bInitDone					: BOOL;
	//arrInitErr					: ARRAY [1..2] OF BOOL;
	//arrInitDone					: ARRAY [1..2] OF BOOL;
	arrSensorScales				: ARRAY [1..10] OF SH_Light.ST_DALI_SensorScaleMode := [	(fMeassureMaxSensor := 1023, fReadMaxSensor := 1023),
																						9(())];
	bCancelHoldTimerOccupancy	: BOOL;
(*	eEventPriorityOccupancy		: E_DALIEventPriority := E_DALIEVENTPRIORITY.Middle;
	nHoldTimerOccupancy			: WORD := 5; // Value in s. 	
	nReportTimerOccupancy		: BYTE := 120; // Value in s, Preset manufacturer value
	nDeadtimeTimerOccupancy		: WORD := 100; // Value in ms, Predefined Value of DALI Standard
	bCancelHoldTimerOccupancy	: BOOL;
	nSensitivityOccupancy		: BYTE:= 3; //setting Sensivity (0..4) 0 (Off), 1 (Min), 2(Low), 3(High) and 4 (Max)

	bEnableLuxEvent				: BOOL;
	eEventPriorityBrightness	: E_DALIEventPriority := E_DALIEVENTPRIORITY.Middle;
	nDeadtimeTimerBrightness	: WORD := 1500; // Value in ms, Predefined Value of DALI Standard
	nHysteresisBrightness		: BYTE := 2; // Value in %
	nHysteresisMinBrightness	: BYTE := 10; // Absolute Value, depending on the manufacturer specific resolution
	nReportTimerBrightness		: BYTE := 120; // Value in s, Preset manufacturer value
*)

	//ModbusComm setup
	
	fbWriteSPLuxLevel			: SH_Light.FB_TwoVal_SelectOne_RTrigChange;
	fbWritePirDelayTIme			: SH_Light.FB_TwoVal_SelectOne_RTrigChange;
	stRoomDataPLC				: SH_Light.ST_RoomDataPLC	:=	(	uiPirOffDelayTime	:= 30,
																	uiSpLuxLevel		:= 500,
																	uiPirDimDelayTime	:= 15,
																	uiSpDimLuxLevel		:= 200
																);
	fbBallastOnHours			: SH_Light.FB_CountOnHours;
	bEnableHourCount			: BOOL := TRUE;
	
	//Non-persistent modbus data
	bPirActive_MB			AT%MX8.0	: BOOL;				//bPirLys i gammel kode
	uiActLuxLevel_MB		AT%MB12		: UINT;				//intHMIAktueltLux i gammel kode
	uiActLightLevelPct_MB	AT%MB16		: UINT;				//intDALI_Gruppe1_Lysniveau i gammel kode
	
	//For Conversion
	uiPirOffMinutes						: UINT;
	udTimeScaling						: UDINT := 60000;
	uiLuxOn								: UINT;
	
	//max values checks
	uiMaxLuxLevel						: UINT := 1023;
	uiMaxPirOffMinutes					: UINT := 180;
	
END_VAR

VAR CONSTANT
	Sensor_DALI_LINE_NUM	: BYTE := 3;
	DALI_LINE_NUM_LIGHT		: BYTE := 2;
	DALI_LINE_NUM_PENDANTS	: BYTE := 0; //0=ingen pendler
END_VAR
VAR PERSISTENT
	stPirSensorData: SH_Light.ST_DALI_Sensor;
	stTuneData: SH_Light.ST_TuneData_EX;
	
	uiPirOffDelayTime_MB	AT%MB10		: UINT;				//ntHMI_Pir_SetValue i gammel kode
	uiSPLuxLevel_MB			AT%MB14		: UINT;				//intHMI_Lux_SetValue i gammel kode
	uiBallastOnHours_MB		AT%MB18		: UINT;				//dintHMILysbraendtimer1 i gammel kode
	byOnHoursOverflowCount				: BYTE;
END_VAR

A_Buttons();
A_LightCtrl();
A_ModbusComm();
A_Sensor();

ACTION A_Buttons:
bTopButtonZone1		:= GVL_EnOcean.strEnOceanSwitch_Rum_4_325.bT2_OFF OR bTopButtonZone1_Visu;
bBottomButtonZone1	:= GVL_EnOcean.strEnOceanSwitch_Rum_4_325.bT2_ON OR bBottomButtonZone1_Visu;
END_ACTION

ACTION A_LightCtrl:

fbLys(
	nZoneID:= 1, 
	bButtonZone1:= bTopButtonZone1,
	bBottomButtonZone1 := bBottomButtonZone1, 
	bButtonZone2:= bButtonZone2, 
	fLuxOn:= fLuxOn, 
	fLuxDim:= fLuxDim, 
	tPIRDim:= tPIRDim, 
	tPIROff:= tPIROff, 
	fOffsetSec:= fOffsetSec, 
	bReInit:= , 
	stDaliSetup:= stDaliSetup, 
	ipCommunication_Prim:= P_DALI_Background.arrfbKL6821Communication[DALI_LINE_NUM_LIGHT], 
	ipCommunication_Sec:= P_DALI_Background.arrfbKL6821Communication[DALI_LINE_NUM_LIGHT], 
	ipCommunication_Supl:= P_DALI_Background.arrfbKL6821Communication[DALI_LINE_NUM_LIGHT], 
	fMinOutputPowerLevelRoom:= 15, 
	fMaxOutputPowerLevelRoom:= 100, 
	nCycleTimeInMS:= SH_Light.DALI_Param.nPlcTaskCycleTimeInMS , 
	bRunTuning:= bRunTuning, 
	bOccupiedRoom=> bOccupiedRoom, 
	bError_Prim=> , 
	nError_Prim=> , 
	stTuneData:=stTuneData , 
	stPirSensorData:= stPirSensorData, 
	stLiveData:= stLiveData);
END_ACTION

ACTION A_ModbusComm:
//Manage data for modbus communication

//Manage data for read-only in PLC
stRoomDataPLC.bPirActive			:= stPirSensorData.bPrc;
stRoomDataPLC.uiActLuxLevel			:= TO_UINT(TRUNC(stPirSensorData.fBrightness));
stRoomDataPLC.uiActLightLevelPct	:= TO_UINT(TRUNC(fbLys.fbBallast.fActlLgtLvl_Prim));
		//stRoomDataPLC.uiActLightLevelPct	:= TO_UINT(TRUNC(fbLys.fbBallast.fActlLgtLvl_Prim)); //if only one group light control
stRoomDataPLC.uiBallastOnHours		:= uiBallastOnHours_MB; //The calculation for BallastOnHours is stored directly to the MB register below


//Assign data for read-only to MB registers
bPirActive_MB			:= stRoomDataPLC.bPirActive;
uiActLuxLevel_MB		:= stRoomDataPLC.uiActLuxLevel;
uiActLightLevelPct_MB	:= stRoomDataPLC.uiActLightLevelPct;

	//calculate BallastOnHours
	fbBallastOnHours(
		bEnableHourCount	:= bEnableHourCount,
		bPauseCount			:= fbLys.fbLightCtrl.bOffZone1,
		uiOnHours			:= uiBallastOnHours_MB,			//OnHours is updated here
		byOverflowCount		:= byOnHoursOverflowCount);


//Manage data for read/write for both PLC and MB registers
fbWriteSPLuxLevel(	nMaxValOut	:= uiMaxLuxLevel,
					nValIn1		:= uiSPLuxLevel_MB,		//nValIn1 takes priotity in case of download or restart
					nValIn2		:= stRoomDataPLC.uiSpLuxLevel,
					nValOut		=> uiLuxOn
				);


fbWritePirDelayTIme(	nMaxValOut	:= uiMaxPirOffMinutes,
						nValIn1		:= uiPirOffDelayTime_MB,		//nValIn1 takes priotity in case of download or restart
						nValIn2		:= stRoomDataPLC.uiPirOffDelayTime,
						nValOut		=> uiPirOffMinutes
					);
					

//Convert read/write modbus data to appropriate datatypes in PLC
fLuxOn	:= TO_REAL(uiLuxOn);			
tPIROff	:= TO_TIME(uiPirOffMinutes*udTimeScaling); //Time conversion defaults to ms

fLuxDim	:= TO_REAL(stRoomDataPLC.uiSpDimLuxLevel);			
tPIRDim	:= TO_TIME(stRoomDataPLC.uiPirDimDelayTime*udTimeScaling); //Time conversion defaults to ms
END_ACTION

ACTION A_Sensor:

fbSensor.ipCommunication := P_DALI_Background.arrfbKL6821Communication[Sensor_DALI_LINE_NUM];


fbSensor(
	byShrtAdr:= bySensorAddr,
	bInitialize:= bInitialize, 
	DALI_LINE_NUM:= Sensor_DALI_LINE_NUM, 
 	//bCancelHoldTimerOccupancy:= bCancelHoldTimerOccupancy, 
	stSensorSetup := stDaliSensorSetup,
	bInitErr=> bInitErr, 
	bInitDone=> bInitDone,
	stPirSensorData:= stPirSensorData, 
	arrSensorScales:= arrSensorScales);

(*
fbSensor(
	arrShrtAdr:= arrSensorAddr,
	bInitialize:= bInitialize, 
	DALI_LINE_NUM:= Sensor_DALI_LINE_NUM, 
 	//bCancelHoldTimerOccupancy:= bCancelHoldTimerOccupancy, 
	stSensorSetup := stDaliSensorSetup,
	arrInitErr=> arrInitErr, 
	arrInitDone=> arrInitDone,
	stPirSensorData:= stPirSensorData, 
	arrSensorScales:= arrSensorScales);
	*)
END_ACTION

END_PROGRAM

// ---- POUs/DALI/DALI_Setup/FBs/FB_Part205Incandescent.TcPOU
FUNCTION_BLOCK FB_Part205Incandescent
VAR_INPUT
	ipDALICommunication					:	I_DALICommunication;
END_VAR
VAR_OUTPUT
	bBusy								:	BOOL;
END_VAR
VAR
	{region "Visu"}
	bReadStatus							:	BOOL;
	bReadParameter						:	BOOL;
	bWrite								:	BOOL;
	sLoadOverCurrentShutdown			:	STRING(5);
	sThermalShutdown					:	STRING(5);
	sOpenCircuitDetection				:	STRING(5);
	sThermalOverload	 				:	STRING(5);
	sInvalidDimmingMethod				:	STRING(5);
	sSupplyVoltageOutOfLimit			:	STRING(5);
	sSupplyFrequencyOutOfLimit			:	STRING(5);
	sLoadVoltageOutOfLimit				:	STRING(5);
	sLoadCurrentOverload				:	STRING(5);
	sLinearDimmingCurve					:	STRING(5);
	sLeadingEdgeModeRunning				:	STRING(5);
	sTrailingEdgeModeRunning			:	STRING(5);
	
	eDimmingCurve						:	Tc3_DALI.E_DALIDimmingCurve;
	{endregion}
		 
	nStep								:	INT;
	nAddress							: 	BYTE;
	bHideWaitSymbol						:	BOOL := TRUE;	
	nFeatures							:	DWORD;
	
	nRmsLoadVoltage						:	BYTE;
	bNoRmsLoadVoltage					:	BOOL;
	fRealLoadPower						:	REAL;
	bNoRealLoadPower					:	BOOL;
	fLoadRating							:	REAL;
	bNoLoadRating						:	BOOL;
	nDimmerTemperature					:	BYTE;
	bNoDimmerTemperature				:	BOOL;
	nRMSSupplyVoltage					:	UINT;
	bNoRMSSupplyVoltage					:	BOOL;
	nRMSLoadCurrent						:	BYTE;
	bNoRMSLoadCurrent					:	BOOL;
	nSupplyFrequency					:	BYTE;
	bNoSupplyFrequency					:	BOOL;
	
	
	bLoadOverCurrentShutdownQueried		:	BOOL;
	bOpenCircuitQueried					:	BOOL;
	bThermalShutdownQueried				:	BOOL;
	bThermalOverloadQueried				:	BOOL;
	bTempQueried						:	BOOL;
	bSupplyVoltageQueried				:	BOOL;
	bSupplyFrequencyQueried				:	BOOL;
	bLoadVoltageQueried					:	BOOL;
	bLoadCurrentQueried					:	BOOL;
	bRealLoadPowerQueried				:	BOOL;
	bLoadRatingQueried					:	BOOL;
	bLoadCurrentOverloadQueried			:	BOOL;
	bDimmingMethodBit0					:	BOOL;
	bDimmingMethodBit1					:	BOOL;
	bNonLogarithmicCurve				:	BOOL;
	bUnsuitableLoadQueried				:	BOOL;
		
	fb103StartQuiescentMode				:	FB_DALI103StartQuiescentMode(0);
	fb103StopQuiescentMode				:	FB_DALI103StopQuiescentMode(0);
	fb205QueryFeatures					:	FB_DALI205QueryFeatures(0);
	
	fb205QueryRMSLoadVoltage			:	FB_DALI205QueryRMSLoadVoltage(0);
	fb205QueryRealLoadPower				:	FB_DALI205QueryRealLoadPower(0);
	fb205QueryLoadRating				:	FB_DALI205QueryLoadRating(0);
	fb205QueryDimmerTemperature			:	FB_DALI205QueryDimmerTemperature(0);
	fb205QueryDimmerStatus				:	FB_DALI205QueryDimmerStatus(0);
	fb205QueryFailureStatus				:	FB_DALI205QueryFailureStatus(0);
	fb205QueryRMSSupplyVoltage			:	FB_DALI205QueryRMSSupplyVoltage(0);
	fb205QueryRMSLoadCurrent			:	FB_DALI205QueryRMSLoadCurrent(0);
	fb205QuerySupplyFrequency			:	FB_DALI205QuerySupplyFrequency(0);
	
	fb205QueryDimmingCurve				:	FB_DALI205QueryDimmingCurve(0);
	fb205SelectDimmingCurve				:	FB_DALI205SelectDimmingCurve(0);
END_VAR

{region "Detect Commands"}
IF (bReadStatus AND (nStep = 0)) THEN
	nStep := 5;
	bReadStatus := FALSE;
	bHideWaitSymbol := FALSE;
END_IF

IF (bReadParameter AND (nStep = 0)) THEN
	nStep := 200;
	bReadParameter := FALSE;
	bHideWaitSymbol := FALSE;
END_IF

IF (bWrite AND (nStep = 0)) THEN
	nStep := 1000;
	bWrite := FALSE;
	bHideWaitSymbol := FALSE;
END_IF
{endregion}
{region "Manage Dialog Selection}
IF (nStep = 0) THEN
	bBusy := FALSE;
ELSE
	bBusy := TRUE;
END_IF
{endregion}

{region "Execute Commands"}
CASE nStep OF
0:
{region "Init"}
	bReadStatus := FALSE;
	bReadParameter := FALSE;
	bHideWaitSymbol := TRUE;

	fb103StartQuiescentMode.ipDALICommunication := ipDALICommunication;
	fb103StopQuiescentMode.ipDALICommunication := ipDALICommunication;
	fb205QueryFeatures.ipDALICommunication := ipDALICommunication;
	fb205QueryDimmingCurve.ipDALICommunication := ipDALICommunication;
	fb205SelectDimmingCurve.ipDALICommunication := ipDALICommunication;
	fb205QueryRMSLoadVoltage.ipDALICommunication := ipDALICommunication;
	fb205QueryRealLoadPower.ipDALICommunication := ipDALICommunication;
	fb205QueryLoadRating.ipDALICommunication := ipDALICommunication;
	fb205QueryDimmerTemperature.ipDALICommunication := ipDALICommunication;
	fb205QueryFailureStatus.ipDALICommunication := ipDALICommunication;
	fb205QueryDimmerStatus.ipDALICommunication := ipDALICommunication;
	fb205QueryRMSSupplyVoltage.ipDALICommunication := ipDALICommunication;
	fb205QueryRMSLoadCurrent.ipDALICommunication := ipDALICommunication;
	fb205QuerySupplyFrequency.ipDALICommunication := ipDALICommunication;
{endregion}
{region "Read Status"}
5:
{region "Start Qiescent Mode"}
	fb103StartQuiescentMode(bStart := TRUE,
							eAddressType := Tc3_DALI.E_DALIAddressType.Broadcast,
							eCommandPriority := Tc3_DALI.E_DALICommandPriority.Middle);
	IF (NOT fb103StartQuiescentMode.bBusy) THEN
		fb103StartQuiescentMode(bStart  := FALSE);
		nStep := 10;
	END_IF
{endregion}
10:
{region "Query Dimmer Features"}
	fb205QueryFeatures(	bStart := TRUE,
						nAddress := nAddress,
						eAddressType := Tc3_DALI.E_DALIAddressType.Short,
						eCommandPriority := Tc3_DALI.E_DALICommandPriority.Middle,
						nFeatures => nFeatures);
	IF (NOT fb205QueryFeatures.bBusy) THEN
	fb205QueryFeatures(bStart := FALSE);
	nStep := 15;
	END_IF
{endregion}
15:
{region "Query RMS Load Voltage"}
	IF (fb205QueryFeatures.nFeatures.11) THEN
		bNoRmsLoadVoltage := FALSE;
		nStep := 20;
	ELSE 
		bNoRmsLoadVoltage := TRUE;
		nStep := 25;
	END_IF
20:
	fb205QueryRMSLoadVoltage(	bStart := TRUE,
								nAddress := nAddress,
								eAddressType := Tc3_DALI.E_DALIAddressType.Short,
								eCommandPriority := Tc3_DALI.E_DALICommandPriority.Middle);
	IF (NOT fb205QueryRMSLoadVoltage.bBusy) THEN
		nRmsLoadVoltage := 2 * (fb205QueryRMSLoadVoltage.nRMSLoadVoltage);
		fb205QueryRMSLoadVoltage(bStart := FALSE);
		nStep := 25;
	END_IF
{endregion}
25:
{region "Query Real Load Power"}
	IF (fb205QueryFeatures.nFeatures.13) THEN
		bNoRealLoadPower := FALSE;
		nStep := 30;
	ELSE
		bNoRealLoadPower := TRUE;
		nStep := 35;
	END_IF
30:
	fb205QueryRealLoadPower(bStart := TRUE,
							nAddress := nAddress,
							eAddressType := Tc3_DALI.E_DALIAddressType.Short,
							eCommandPriority := Tc3_DALI.E_DALICommandPriority.Middle);
	IF (NOT fb205QueryRealLoadPower.bBusy) THEN
		fRealLoadPower := TO_REAL(fb205QueryRealLoadPower.nRealLoadPower / 4);
		fb205QueryRealLoadPower(bStart := FALSE);
		nStep := 35;
	END_IF
{endregion}
35:
{region "Query Load Rating"}
	IF (fb205QueryFeatures.nFeatures.14) THEN
		bNoLoadRating := FALSE;
		nStep := 40;
	ELSE
		bNoLoadRating := TRUE;
		nStep := 45;
	END_IF
40:
	fb205QueryLoadRating(	bStart := TRUE,
							nAddress := nAddress,
							eAddressType := Tc3_DALI.E_DALIAddressType.Short,
							eCommandPriority := Tc3_DALI.E_DALICommandPriority.Middle);
	IF (NOT fb205QueryLoadRating.bBusy) THEN
		fLoadRating := TO_REAL( fb205QueryLoadRating.nLoadRating) * 0.15;
		fb205QueryLoadRating(bStart := FALSE);
		nStep := 45;
	END_IF
{endregion}
45:
{region "Query Dimmer Temperature"} 
	IF (fb205QueryFeatures.nFeatures.8) THEN
		bNoDimmerTemperature := FALSE;
		nStep := 50;
	ELSE 
		bNoDimmerTemperature := TRUE;
		nStep := 55;
	END_IF
50:
	fb205QueryDimmerTemperature(bStart := TRUE,
								nAddress := nAddress,
								eAddressType := Tc3_DALI.E_DALIAddressType.Short,
								eCommandPriority := Tc3_DALI.E_DALICommandPriority.Middle);
	IF (NOT fb205QueryDimmerTemperature.bBusy) THEN
		nDimmerTemperature := (fb205QueryDimmerTemperature.nDimmerTemperature - 40);
		fb205QueryDimmerTemperature(bStart := FALSE);
		nStep := 55;
	END_IF
{endregion}
55:
{region "Query RMS Supply Voltage"}
	IF (fb205QueryFeatures.nFeatures.9) THEN
		bNoRMSSupplyVoltage := FALSE;
		nStep := 60;
	ELSE 
		bNoRMSSupplyVoltage := TRUE;
		nStep := 65;
	END_IF
60:
	fb205QueryRMSSupplyVoltage(	bStart := TRUE,
								nAddress := nAddress,
								eAddressType := Tc3_DALI.E_DALIAddressType.Short,
								eCommandPriority := Tc3_DALI.E_DALICommandPriority.Middle);
	IF (NOT fb205QueryRMSSupplyVoltage.bBusy) THEN
		nRMSSupplyVoltage := ( fb205QueryRMSSupplyVoltage.nRMSSupplyVoltage * 2);
		fb205QueryRMSSupplyVoltage(bStart := FALSE);
		nStep := 65;
	END_IF
{endregion}
65:
{region "Query RMS Load Current"}
	IF (fb205QueryFeatures.nFeatures.12) THEN
		bNoRMSLoadCurrent := FALSE;
		nStep := 70;
	ELSE 
		bNoRMSLoadCurrent := TRUE;
		nStep := 75;
	END_IF
70:
	fb205QueryRMSLoadCurrent(	bStart := TRUE,
								nAddress := nAddress,
								eAddressType := Tc3_DALI.E_DALIAddressType.Short,
								eCommandPriority := Tc3_DALI.E_DALICommandPriority.Middle,
								nRMSLoadCurrent => nRMSLoadCurrent);
	IF (NOT fb205QueryRMSLoadCurrent.bBusy) THEN
		nRMSLoadCurrent := (fb205QueryRMSLoadCurrent.nRMSLoadCurrent / 2);
		fb205QueryRMSSupplyVoltage(bStart := FALSE);
		nStep := 75;
	END_IF
{endregion}
75:
{region "Query Supply Frequency"}
	IF (fb205QueryFeatures.nFeatures.10) THEN
		bNoSupplyFrequency := FALSE;
		nStep := 80;
	ELSE
		bNoSupplyFrequency := TRUE;
		nStep := 90;
	END_IF
80:
	fb205QuerySupplyFrequency(	bStart := TRUE,
								nAddress := nAddress,
								eAddressType := Tc3_DALI.E_DALIAddressType.Short,
								eCommandPriority := Tc3_DALI.E_DALICommandPriority.Middle);
	IF (NOT fb205QuerySupplyFrequency.bBusy) THEN
		nSupplyFrequency := (fb205QuerySupplyFrequency.nSupplyFrequency / 2);
		fb205QuerySupplyFrequency(bStart := FALSE);
		nStep := 90;
	END_IF
{endregion}
90:
{region "Query Failure Status"}
	fb205QueryFailureStatus(	bStart := TRUE,
								nAddress := nAddress,
								eAddressType := Tc3_DALI.E_DALIAddressType.Short,
								eCommandPriority := Tc3_DALI.E_DALICommandPriority.Middle);
	IF (NOT fb205QueryFailureStatus.bBusy) THEN
		fb205QueryFailureStatus(bStart := FALSE);
		sLoadOverCurrentShutdown := SEL(fb205QueryFailureStatus.nFailureStatus.0, 'False', 'True');
		sOpenCircuitDetection := SEL(fb205QueryFailureStatus.nFailureStatus.1, 'False', 'True');
		sThermalShutdown := SEL(fb205QueryFailureStatus.nFailureStatus.5, 'False', 'True');
		sThermalOverload := SEL(fb205QueryFailureStatus.nFailureStatus.6, 'False', 'True');
		sInvalidDimmingMethod := SEL(fb205QueryFailureStatus.nFailureStatus.8, 'False', 'True');
		sSupplyVoltageOutOfLimit := SEL(fb205QueryFailureStatus.nFailureStatus.9, 'False', 'True');
		sSupplyFrequencyOutOfLimit := SEL(fb205QueryFailureStatus.nFailureStatus.10, 'False', 'True');
		sLoadVoltageOutOfLimit := SEL(fb205QueryFailureStatus.nFailureStatus.11, 'False', 'True');
		sLoadCurrentOverload := SEL(fb205QueryFailureStatus.nFailureStatus.12, 'False', 'True');
		nStep := 100;
	END_IF
{endregion}
100:
{region "Query Dimmer Status"}
	fb205QueryDimmerStatus(	bStart := TRUE,
							nAddress := nAddress,
							eAddressType := Tc3_DALI.E_DALIAddressType.Short,
							eCommandPriority := Tc3_DALI.E_DALICommandPriority.Middle);
	IF (NOT fb205QueryDimmerStatus.bBusy) THEN
		fb205QueryDimmerStatus(bStart := FALSE);
		sLeadingEdgeModeRunning := SEL(fb205QueryDimmerStatus.nDimmerStatus.0, 'False', 'True');
		sTrailingEdgeModeRunning := SEL(fb205QueryDimmerStatus.nDimmerStatus.1, 'False', 'True');
		sLinearDimmingCurve := SEL(fb205QueryDimmerStatus.nDimmerStatus.4, 'False', 'True');
		nStep := 110;
	END_IF
{endregion}
110:
{region "Stop Qiescent Mode"}
	fb103StopQuiescentMode(	bStart := TRUE,
							eAddressType := Tc3_DALI.E_DALIAddressType.Broadcast,
							eCommandPriority := Tc3_DALI.E_DALICommandPriority.Middle);
	IF (NOT fb103StopQuiescentMode.bBusy) THEN
		fb103StopQuiescentMode(bStart := FALSE);
		nStep := 0;
	END_IF
{endregion}
{endregion}

{region "Read Parameter"}
200:
{region "Start Qiescent Mode"}
	fb103StartQuiescentMode(bStart := TRUE,
							eAddressType := Tc3_DALI.E_DALIAddressType.Broadcast,
							eCommandPriority := Tc3_DALI.E_DALICommandPriority.Middle);
	IF (NOT fb103StartQuiescentMode.bBusy) THEN
		fb103StartQuiescentMode(bStart := FALSE);
		nStep := 210;
	END_IF
{endregion}
210:
{region "Query Dimmer Features"}
	fb205QueryFeatures(	bStart := TRUE,
						nAddress := nAddress,
						eAddressType := Tc3_DALI.E_DALIAddressType.Short,
						eCommandPriority := Tc3_DALI.E_DALICommandPriority.Middle,
						nFeatures => nFeatures);
	IF (NOT fb205QueryFeatures.bBusy) THEN
		fb205QueryFeatures(bStart := FALSE);
		bLoadOverCurrentShutdownQueried := nFeatures.0;
		bOpenCircuitQueried := nFeatures.1;
		bThermalShutdownQueried := nFeatures.5;
		bThermalOverloadQueried := nFeatures.6;
		bTempQueried := nFeatures.8;
		bSupplyVoltageQueried := nFeatures.9;
		bSupplyFrequencyQueried := nFeatures.10;
		bLoadVoltageQueried := nFeatures.11;
		bLoadCurrentQueried := nFeatures.12;
		bRealLoadPowerQueried := nFeatures.13;
		bLoadRatingQueried := nFeatures.14;
		bLoadCurrentOverloadQueried := nFeatures.15;
		bDimmingMethodBit0 := nFeatures.16;
		bDimmingMethodBit1 := nFeatures.17;
		bNonLogarithmicCurve := nFeatures.19;
		bUnsuitableLoadQueried := nFeatures.23;
		nStep := 220;
	END_IF
{endregion}
220:
{region "Query Dimming Curve"}
	fb205QueryDimmingCurve(	bStart := TRUE,
							nAddress := nAddress,
							eAddressType := Tc3_DALI.E_DALIAddressType.Short,
							eCommandPriority := Tc3_DALI.E_DALICommandPriority.Middle);
	IF (NOT fb205QueryDimmingCurve.bBusy) THEN
		fb205QueryDimmingCurve(	bStart := FALSE);
		eDimmingCurve := fb205QueryDimmingCurve.eDimmingCurve;
		nStep := 230;
	END_IF
{endregion}
230:
{region "Stop Qiescent Mode"}
	fb103StopQuiescentMode(	bStart := TRUE,
							eAddressType := Tc3_DALI.E_DALIAddressType.Broadcast,
							eCommandPriority := Tc3_DALI.E_DALICommandPriority.Middle);
	IF (NOT fb103StopQuiescentMode.bBusy) THEN
		fb103StopQuiescentMode(bStart := FALSE);
		nStep := 0;
	END_IF
{endregion}
{endregion}

{region "Write Parameter"}
1000:
	fb205SelectDimmingCurve(bStart := TRUE,
							nAddress := nAddress,
							eAddressType := Tc3_DALI.E_DALIAddressType.Short,
							eCommandPriority := Tc3_DALI.E_DALICommandPriority.Middle,
							eDimmingCurve := eDimmingCurve);
	IF (NOT fb205SelectDimmingCurve.bBusy) THEN
		fb205SelectDimmingCurve.bStart := FALSE;
		nStep := 0;
	END_IF
{endregion}
END_CASE

END_FUNCTION_BLOCK

// ---- POUs/DALI/PRGs/EnergyData/P_DALI_Energy_Line_old.TcPOU
(*
EnergyReporting reads ActiveEnergy (part 252) for all present ballasts on all (configured) DALI-lines where GVL_DALI.g_arrEnergyData[*DALI-line*,*ballast*].bHasEnergyData is TRUE.
Results are stored in GVL_DALI.g_arrEnergyData[*DALI-line*,*ballast*].fActiveEnergy. Energy Data for individual ballasts is NOT persistent.
The engergy sum per DALI-Line (Wh) and Total Energy (kWh) are persistent.

If bCheckActiveEnergy is TRUE, all present ballasts are queried for ActiveEnergy and bHasEnergyData is updated accordingly.
This will result in errors for any ballast that does not comply with part 252.
Errors will not be triggered for activations where bCheckActiveEnergy is FALSE.

After shutdown or download to PLC EnergyReporting is activated automatically internally with bCheckActiveEnergy set to TRUE

EnergyReporting is activated automatically at TOD 0:00, 6:00, 12:00, 18:00 (configurable)

NB:	The priority of commands are set to "middle" internally. Updating all lines will take a couple of minutes to finish, so be patient.
	Other critical commands on the DALI-lines take priotity.
	Add appropriate communication immediately after configuration of a new KL6821 terminal.
	That is, arrfbDALI_EnergyReporting[*DALI-Line*].ipDALICommunication := P_DALI_Background.arrfbKL6821Communication[*DALI-Line*];
*)


PROGRAM P_DALI_Energy_Line_old
VAR
	arrfbDALI_EnergyReporting	: ARRAY[1..SH_Light.DALI_Param.MAX_DALIV2_LINES] OF FB_DALI_EnergyReporting_Test;
	bReadEnergyDataAllLines		: BOOL;
	arrReadEnergyData			: ARRAY[1..SH_Light.DALI_Param.MAX_DALIV2_LINES] OF BOOL;
	arrCheckActiveEnergy		: ARRAY[1..SH_Light.DALI_Param.MAX_DALIV2_LINES] OF BOOL;
	arrDone						: ARRAY[1..SH_Light.DALI_Param.MAX_DALIV2_LINES] OF BOOL;
	arrfbRTrigDone				: ARRAY[1..SH_Light.DALI_Param.MAX_DALIV2_LINES] OF R_TRIG;
	arrRTrigDone				: ARRAY[1..SH_Light.DALI_Param.MAX_DALIV2_LINES] OF BOOL;
	
	byEnergyLineIdx: BYTE;
	
	//variables to store persistent data correctly
	byCount								: BYTE;
	nMaxControlGearOperatingTimeTmp		: ARRAY[1..SH_Light.DALI_Param.MAX_DALIV2_LINES] OF UDINT;
	nMaxControlGearOperatingTime		: ARRAY[1..SH_Light.DALI_Param.MAX_DALIV2_LINES] OF UDINT;
	nMaxControlGearOperatingHoursTmp	: UINT;
	//byShrtAddrOfMostUsedBallast		: ARRAY[1..SH_Light.DALI_Param.MAX_DALIV2_LINES] OF BYTE;
	arrDaliLineEnergySumWH_Tmp			: ARRAY[1..SH_Light.DALI_Param.MAX_DALIV2_LINES] OF LREAL;
	arrDaliLineEnergySumWH_Old			: ARRAY[1..SH_Light.DALI_Param.MAX_DALIV2_LINES] OF LREAL;
	arrDaliLineEnergyChangeWH			: ARRAY[1..SH_Light.DALI_Param.MAX_DALIV2_LINES] OF LREAL;
	nTotalEnergyKWHTmp					: UINT;
	fMaxEnergyValueTrust				: LREAL := 1000000000;
	nMaxTimeValueTrust					: UDINT := 100000000;
	
	//Task scheduling
	stLocalSystemTime 		: TIMESTRUCT;
	fbLocalSystemTime 		: FB_LocalSystemTime;
	bGetTime 				: BOOL := TRUE;
	tTimeOut 				: TIME := DEFAULT_ADS_TIMEOUT;
	bLocalSystemTimeValid	: BOOL;
	tzID       				: E_TimeZoneID := eTimeZoneID_Invalid;
	
	tdSystemTime			: TOD;
	btestTodCompare			: BOOL;
	
	
END_VAR
VAR CONSTANT
	tdMidnight						: TOD := TOD#0:0:0;
	tdMorning						: TOD := TOD#6:0:0;
	tdMidDay						: TOD := TOD#12:0:0;
	tdEvening						: TOD := TOD#18:0:0;
	tCheckDuration					: TIME:= T#5S;
	tdTestsum						: TOD := (tdMidnight + tCheckDuration);
END_VAR

VAR PERSISTENT
	arrDaliLineEnergySumWH				: ARRAY[1..SH_Light.DALI_Param.MAX_DALIV2_LINES] OF LREAL;
	nTotalEnergykWH						: UINT;
	nMaxControlGearOperatingHours		: UINT;
END_VAR


arrfbDALI_EnergyReporting[1].ipDALICommunication := P_DALI_Background.arrfbKL6821Communication[1];
arrfbDALI_EnergyReporting[2].ipDALICommunication := P_DALI_Background.arrfbKL6821Communication[2];
arrfbDALI_EnergyReporting[3].ipDALICommunication := P_DALI_Background.arrfbKL6821Communication[3];
arrfbDALI_EnergyReporting[4].ipDALICommunication := P_DALI_Background.arrfbKL6821Communication[4];
//arrfbDALI_EnergyReporting[5].ipDALICommunication := P_DALI_Background.arrfbKL6821Communication[5];
//arrfbDALI_EnergyReporting[6].ipDALICommunication := P_DALI_Background.arrfbKL6821Communication[6]; // for more update SH_Light.DALI_Param.MAX_DALIV2_LINES


fbLocalSystemTime(
	sNetID:= '', 
	bEnable:= bGetTime, 
	dwCycle:= 2, // cycle time (in seconds) , Synchronization  every 2 seconds.
	dwOpt:= 1, //Bit 0: If this is set, the Windows system time is additionally synchronized cyclically with the hardware clock (RTC) (corresponds to the function NT_SetTimeToRTCTime).
	tTimeout:= tTimeOut, 
	bValid=> bLocalSystemTimeValid, 
	systemTime=> stLocalSystemTime, 
	tzID=> tzID);
	
tdSystemTime := SYSTEMTIME_TO_TOD(systemTime := stLocalSystemTime);
IF	((tdSystemTime > tdMidnight AND tdSystemTime < (tdMidnight + tCheckDuration)) OR (tdSystemTime > tdMorning AND tdSystemTime < (tdMorning + tCheckDuration)) OR
	(tdSystemTime > tdMidDay AND tdSystemTime < (tdMidDay + tCheckDuration)) OR (tdSystemTime > tdEvening AND tdSystemTime < (tdEvening + tCheckDuration))) THEN
	bReadEnergyDataAllLines := TRUE;
END_IF

FOR byEnergyLineIdx := 1 TO SH_Light.DALI_Param.MAX_DALIV2_LINES DO
	IF bReadEnergyDataAllLines = TRUE THEN
		arrReadEnergyData[byEnergyLineIdx] := TRUE;
	END_IF;
	arrfbDALI_EnergyReporting[byEnergyLineIdx](
		bExecute:= arrReadEnergyData[byEnergyLineIdx], 
		DALI_LINE_NUM:= byEnergyLineIdx,
		bCheckActiveEnergy := arrCheckActiveEnergy[byEnergyLineIdx],
		bBusy=> , 
		bActionBusy=> , 
		bErr=>, 
		nErrorId=> ,
		bDone =>  arrDone[byEnergyLineIdx]);
	arrfbRTrigDone[byEnergyLineIdx](CLK := arrDone[byEnergyLineIdx], Q => arrRTrigDone[byEnergyLineIdx]);
	IF arrRTrigDone[byEnergyLineIdx] THEN
		bReadEnergyDataAllLines := FALSE;
		arrReadEnergyData[byEnergyLineIdx] := FALSE;
		nMaxControlGearOperatingTime[byEnergyLineIdx] := 0;
		FOR byCount := 1 TO 63 DO
			IF SH_Light.GVL_DALI.g_arrEnergyData[byEnergyLineIdx, byCount].fActiveEnergy < fMaxEnergyValueTrust THEN
			arrDaliLineEnergySumWH_Tmp[byEnergyLineIdx] := arrDaliLineEnergySumWH_Tmp[byEnergyLineIdx] + SH_Light.GVL_DALI.g_arrEnergyData[byEnergyLineIdx, byCount].fActiveEnergy;
			END_IF
			IF SH_Light.GVL_DALI.g_arrEnergyData[byEnergyLineIdx, byCount].nControlGearOperatingTime < nMaxTimeValueTrust THEN
			nMaxControlGearOperatingTimeTmp[byEnergyLineIdx] := MAX(nMaxControlGearOperatingTimeTmp[byEnergyLineIdx], SH_Light.GVL_DALI.g_arrEnergyData[byEnergyLineIdx, byCount].nControlGearOperatingTime);
			END_IF
			IF byCount = 63 THEN
				arrDaliLineEnergySumWH_Old[byEnergyLineIdx] := arrDaliLineEnergySumWH[byEnergyLineIdx];
				arrDaliLineEnergySumWH[byEnergyLineIdx] := arrDaliLineEnergySumWH_Tmp[byEnergyLineIdx];
				arrDaliLineEnergyChangewH[byEnergyLineIdx] := arrDaliLineEnergySumWH[byEnergyLineIdx] - arrDaliLineEnergySumWH_Old[byEnergyLineIdx];
				IF arrDaliLineEnergyChangeWH[byEnergyLineIdx] < 0 THEN
					arrDaliLineEnergyChangeWH[byEnergyLineIdx] := 0;
				END_IF
				nTotalEnergyKWHTmp := TO_UINT(TRUNC((arrDaliLineEnergySumWH_Old[byEnergyLineIdx] + arrDaliLineEnergyChangeWH[byEnergyLineIdx])*EXPT(10,-3))); //The line above checks for for negative values. As so the conversion to UINT is appropriate.
				arrDaliLineEnergySumWH_Tmp[byEnergyLineIdx] := 0;
				nMaxControlGearOperatingTime[byEnergyLineIdx] := nMaxControlGearOperatingTimeTmp[byEnergyLineIdx];
				nMaxControlGearOperatingTimeTmp[byEnergyLineIdx] := 0;
			END_IF
		END_FOR
	END_IF 
	nMaxControlGearOperatingHoursTmp := MAX(nMaxControlGearOperatingHoursTmp, TO_UINT(TRUNC(nMaxControlGearOperatingTime[byEnergyLineIdx]*EXPT(60,-2)))); //Maximum of positive numbers are positive. As so the conversion to UINT is appropriate.	
END_FOR;
nMaxControlGearOperatingHours := nMaxControlGearOperatingHoursTmp;
nTotalEnergykWH := nTotalEnergyKWHTmp;

GVL_AHDataModbus.nMaxControlGearOperatingHours := nMaxControlGearOperatingHours;
GVL_AHDataModbus.nTotalEnergyKWH := nTotalEnergykWH;
(*
fDaliLineEnergySum[1]			:= 0;
fDaliLineEnergySum[2]			:= 0;
fDaliLineEnergySum[3]			:= 0;
fDaliLineEnergySum[4]			:= 0;
nTotalEnergyKWH					:= 0;
nMaxControlGearOperatingHours	:= 0;
*)

END_PROGRAM

// ---- POUs/EnOcean/P_EnOcean.TcPOU
PROGRAM P_EnOcean
VAR
	fbKL6581			: FB_KL6581;
	stKL6581_in  AT %I* : KL6581_INPUT;
	stKL6581_out AT %Q*	: KL6581_OUTPUT;
	stKL6581			: STR_KL6581;
	bInitCom			: BOOL := TRUE;
	
	arrEnOcean_Search	: ARRAY [1..8] OF FB_EnOcean_Search;
	nSearchIdx			: BYTE;
	bSerach				: BOOL;
	arrDevices			: ARRAY [1..8] OF INT;
	arrID				: ARRAY [1..8, 0..255] OF DWORD;
	
		//Trykknapper Atrium
	fbGang_3_109_Kantine_Tryk_PladeA	: FB_Rec_RPS_Switch;
	fbAtriumNiveau_Tryk_PladeB				: FB_Rec_RPS_Switch;
	fbAtriumNiveau_Tryk_Sevice				: FB_Rec_RPS_Switch;			

	//Trykknapper på gange
	fbGang_4_313_Tryk_Indgang					: FB_Rec_RPS_Switch;
	fbGang_4_313_Tryk_Pendler					: FB_Rec_RPS_Switch;
	
	//Trykknapper i rum
	fbRum_3_329_Tryk_Indgang					: FB_Rec_RPS_Switch;
	fbRum_3_329_Tryk_Tavle						: FB_Rec_RPS_Switch;
	fbRum_4_307_Tryk_Indgang					: FB_Rec_RPS_Switch;
	fbRum_4_307_Tryk_Pendler					: FB_Rec_RPS_Switch;
	fbRum_4_311_Tryk							: FB_Rec_RPS_Switch;
	fbRum_4_313_Tryk							: FB_Rec_RPS_Switch;
	fbRum_4_316_Tryk							: FB_Rec_RPS_Switch;
	fbRum_4_317_Tryk							: FB_Rec_RPS_Switch;
	fbRum_4_321_Tryk							: FB_Rec_RPS_Switch;
	fbRum_4_322_Tryk							: FB_Rec_RPS_Switch;
	
END_VAR

VAR CONSTANT
	byNode_1: BYTE := 1;
	byNode_2: BYTE := 2;
	byNode_3: BYTE := 3;
	byNode_4: BYTE := 4;
	byNode_5: BYTE := 5;
	byNode_6: BYTE := 6;
	byNode_7: BYTE := 7;
	byNode_8: BYTE := 8;
END_VAR


(* Kommunikation mit der KL6581. *)
(* Communication with the KL6581. *)
fbKL6581(
	bInit			:= bInitCom,
	nIdx			:= 2,
	stKL6581_in		:= stKL6581_In,
	stKL6581_out	:= stKL6581_Out,
	bReady			=> ,
	bBusy			=> ,
	bError			=> ,
	iErrorID		=> ,
	str_KL6581		=> stKL6581);

GVL_AHDataModbus.EnOceanError	:= TO_UINT(fbKL6581.iErrorID);

(* Warten bis der Kommunikationsbaustein initialisiert wurde.*)
(* Wait until the communication function block has been initialized. *)
IF (NOT fbKL6581.bReady) THEN
	RETURN;
END_IF

FOR nSearchIdx:= 1 TO 8 DO
	arrEnOcean_Search[nSearchIdx](
		bStart:= TRUE, 
		str_KL6581:= stKL6581 , 
		byNode:= nSearchIdx, 
		bReceive=> , 
		iDevices=>arrDevices[nSearchIdx] , 
		ar_ID=> );
		
		MEMCPY(ADR(arrID[nSearchIdx,0]), ADR(arrEnOcean_Search[nSearchIdx].ar_ID), SIZEOF(arrEnOcean_Search[nSearchIdx].ar_ID)); 
END_FOR

A_Gang_4_313();

A_Rum_3_329();
A_Rum_4_307();
A_Rum_4_311();
A_Rum_4_313();
A_Rum_4_316();
A_Rum_4_317();
A_Rum_4_321();
A_Rum_4_322();
//AtriumNiveau
A_AtriumNiveau();

ACTION A_AtriumNiveau:
fbAtriumNiveau_Tryk_PladeB(
	str_KL6581:=stKL6581 , 
	byNode:=0, 
	dw_ID:= 16#0029B92D, 
	str_EnOceanSwitch=> GVL_EnOcean.strEnOceanSwitch_AtriumNiveau_PladeB,
	by_Node=> , 
	bReceive=> );
(*
fbAtriumNiveau_Tryk_Sevice(
	str_KL6581:=stKL6581 , 
	byNode:=0, 
	dw_ID:= 16#00FEE4FE87, 
	str_EnOceanSwitch=> GVL_EnOcean.strEnOceanSwitch_AtriumNiveau_Service, 
	by_Node=> , 
	bReceive=> );
*)
END_ACTION

ACTION A_Gang_4_313:
fbGang_4_313_Tryk_Indgang(
	str_KL6581:=stKL6581 , 
	byNode:=byNode_2 , 
	dw_ID:= 16#0029AD03, 
	str_EnOceanSwitch=> GVL_EnOcean.strEnOceanSwitch_Gang_4_313_Indgang, 
	by_Node=> , 
	bReceive=> );
	
fbGang_4_313_Tryk_Pendler(
	str_KL6581:=stKL6581 , 
	byNode:=byNode_2 , 
	dw_ID:= 16#003C1D2B, 
	str_EnOceanSwitch=> GVL_EnOcean.strEnOceanSwitch_Gang_4_313_Pendler, 
	by_Node=> , 
	bReceive=> );
END_ACTION

ACTION A_Rum_3_329:
fbRum_3_329_Tryk_Indgang(
	str_KL6581:=stKL6581 , 
	byNode:=byNode_2 , 
	dw_ID:= 16#0029AD0B, 
	str_EnOceanSwitch=> GVL_EnOcean.strEnOceanSwitch_Rum_3_329_Indgang, 
	by_Node=> , 
	bReceive=> );

fbRum_3_329_Tryk_Tavle(
	str_KL6581:=stKL6581 , 
	byNode:=byNode_2 , 
	dw_ID:= 16#0029AD2B, 
	str_EnOceanSwitch=> GVL_EnOcean.strEnOceanSwitch_Rum_3_329_Tavle, 
	by_Node=> , 
	bReceive=> );
END_ACTION

ACTION A_Rum_4_307:
fbRum_4_307_Tryk_Indgang(
	str_KL6581:=stKL6581 , 
	byNode:=byNode_2 , 
	dw_ID:= 16#0029AD0E, 
	str_EnOceanSwitch=> GVL_EnOcean.strEnOceanSwitch_Rum_4_307_Indgang, 
	by_Node=> , 
	bReceive=> );
	
	fbRum_4_307_Tryk_Pendler(
	str_KL6581:=stKL6581 , 
	byNode:=byNode_2 , 
	dw_ID:= 16#0029AD5E, 
	str_EnOceanSwitch=> GVL_EnOcean.strEnOceanSwitch_Rum_4_307_Pendler, 
	by_Node=> , 
	bReceive=> );
END_ACTION

ACTION A_Rum_4_311:
fbRum_4_311_Tryk(
	str_KL6581:=stKL6581 , 
	byNode:=byNode_2 , 
	dw_ID:= 16#0029AD65, 
	str_EnOceanSwitch=> GVL_EnOcean.strEnOceanSwitch_Rum_4_311, 
	by_Node=> , 
	bReceive=> );
END_ACTION

ACTION A_Rum_4_313:
fbRum_4_313_Tryk(
	str_KL6581:=stKL6581 , 
	byNode:=byNode_2 , 
	dw_ID:= 16#0029AD3D, 
	str_EnOceanSwitch=> GVL_EnOcean.strEnOceanSwitch_Rum_4_313, 
	by_Node=> , 
	bReceive=> );
END_ACTION

ACTION A_Rum_4_316:
fbRum_4_316_Tryk(
	str_KL6581:=stKL6581 , 
	byNode:=byNode_2 , 
	dw_ID:= 16#0029AD3B, 
	str_EnOceanSwitch=> GVL_EnOcean.strEnOceanSwitch_Rum_4_316, 
	by_Node=> , 
	bReceive=> );
END_ACTION

ACTION A_Rum_4_317:
fbRum_4_317_Tryk(
	str_KL6581:=stKL6581 , 
	byNode:=byNode_2 , 
	dw_ID:= 16#29AD58, 
	str_EnOceanSwitch=> GVL_EnOcean.strEnOceanSwitch_Rum_4_317, 
	by_Node=> , 
	bReceive=> );
END_ACTION

ACTION A_Rum_4_321:
fbRum_4_321_Tryk(
	str_KL6581:=stKL6581 , 
	byNode:=byNode_2 , 
	dw_ID:= 16#FEE4ED58, 
	str_EnOceanSwitch=> GVL_EnOcean.strEnOceanSwitch_Rum_4_321, 
	by_Node=> , 
	bReceive=> );
END_ACTION

ACTION A_Rum_4_322:
fbRum_4_322_Tryk(
	str_KL6581:=stKL6581 , 
	byNode:=byNode_2 , 
	dw_ID:= 16#0029AD45, 
	str_EnOceanSwitch=> GVL_EnOcean.strEnOceanSwitch_Rum_4_322, 
	by_Node=> , 
	bReceive=> );
END_ACTION

END_PROGRAM

// ---- POUs/MAIN.TcPOU
PROGRAM MAIN
VAR
	nAlive: INT;
	breset: BOOL;
	nDemoVariable : INT;
	nCX8200_State	AT %I*	: UINT;
END_VAR

VAR PERSISTENT
	nDemoVar_Persist: INT;
END_VAR

nAlive:= nAlive + 1;
GVL_AHDataModbus.nCX8200_State_MB := nCX8200_State;

P_SystemDK.M_nCyclic(bReset := breset );
P_DALI_DIAG();
			//P_EnOcean(); Testing fast task
DALI_Commissioning();
P_DALI_Background();


P_DALI_Energy_Line();
P_AHModbusComm();

//Gange
P_Gang_4_308();
P_Gang_4_310A();
P_Gang_4_313();
P_gang_3_309();

//Rum
P_Rum_3_329();
P_Rum_4_307();
P_Rum_4_311();
P_Rum_4_313();
P_Rum_4_316();
P_Rum_4_317();
P_Rum_4_321();
P_Rum_4_322();


//P_DALI_Energy_Firmware_Test();

END_PROGRAM

// ---- GlobalTextList.TcGTLO
TEXTLIST GlobalTextList
  621 = '%d'
  6 = 'Bottom Button'
  482 = 'Button 1'
  720 = 'Button 2'
  1902 = 'DALI Line:'
  1180 = 'DI1 falling edge'
  1218 = 'DI1 rising edge'
  1726 = 'DI2 falling edge'
  1876 = 'DI2 rising edge'
  519 = 'Dim Dwn'
  63 = 'Dim Up'
  2135 = 'Do not lock process image in case of \nDALI commands from DI1 or DI2'
  967 = 'Gang 1.312A'
  256 = 'Gang 1.315'
  906 = 'Gang 1.316'
  207 = 'Gang 2.344'
  66 = 'Gang 2.344A'
  583 = 'Gang 2.350'
  985 = 'Gang 3.362A'
  67 = 'Gang 3.363A'
  173 = 'Gang 3.363B'
  406 = 'Gang 4.308'
  712 = 'Gang 4.310A'
  692 = 'Gang 4.313'
  524 = 'Gang 6.310'
  316 = 'Gang 7.301'
  492 = 'Internal DALI power supply disabled'
  1771 = 'K-Bus Watchdog'
  1811 = 'Lockable bytes: changeable if "Offset 2" has the Value 85 (0x55).\nFor changing use decimal value.'
  43 = 'Lys Auto'
  444 = 'Lys Rum'
  489 = 'Lys Zone 1'
  2046 = 'Memory Bank:'
  23 = 'Name'
  926 = 'Name of byte in memory bank'
  22 = 'Offset'
  1329 = 'Offset in memory bank'
  708 = 'PIR'
  457 = 'PIR status'
  373 = 'Read'
  2418 = 'Reset inactive process image'
  874 = 'Rum 1.106'
  65 = 'Rum 1.108'
  175 = 'Rum 1.111A'
  924 = 'Rum 1.111C'
  219 = 'Rum 1.111D'
  690 = 'Rum 1.111E'
  912 = 'Rum 1.115'
  126 = 'Rum 1.118'
  215 = 'Rum 1.312A'
  725 = 'Rum 1.318'
  839 = 'Rum 1.319'
  456 = 'Rum 1.320'
  800 = 'Rum 1.321'
  622 = 'Rum 1.322'
  646 = 'Rum 1.323'
  966 = 'Rum 1.324'
  95 = 'Rum 1.325'
  335 = 'Rum 1.326'
  150 = 'Rum 1.327'
  651 = 'Rum 1.328'
  980 = 'Rum 1.330'
  262 = 'Rum 1115'
  642 = 'Rum 2.341'
  978 = 'Rum 2.345'
  736 = 'Rum 2.349'
  593 = 'Rum 2.351'
  122 = 'Rum 2.352'
  27 = 'Rum 2.353'
  41 = 'Rum 2.354'
  697 = 'Rum 2.355'
  826 = 'Rum 2.356'
  561 = 'Rum 2.357'
  952 = 'Rum 3.329'
  623 = 'Rum 3_329'
  174 = 'Rum 4.307'
  166 = 'Rum 4.311'
  870 = 'Rum 4.313'
  584 = 'Rum 4.316'
  812 = 'Rum 4.317'
  458 = 'Rum 4.321'
  565 = 'Rum 4.322'
  803 = 'Rum 4.324'
  430 = 'Rum 6.310 Sofagruppe'
  348 = 'Rum 6.327'
  891 = 'Rum 6.328'
  11 = 'Rum 6.329'
  72 = 'Rum 6.330B'
  197 = 'Rum 6.331'
  564 = 'Rum 6.333'
  997 = 'Rum 6.337'
  31 = 'Rum 6_330A'
  1041 = 'Short Address:'
  395 = 'SP_Lux: %.0f'
  525 = 'SP_Lux: %f'
  2458 = 'Terminal Event'
  849 = 'Test Type A'
  973 = 'Top Button'
  24 = 'Value Dec'
  1435 = 'Value decimal'
  25 = 'Value Hex'
  2231 = 'Value hexadecimal,\nto change use\nvalue decimal'
  374 = 'Write'
  1047 = 'Write default values'
  490 = 'Write parameters'
END_TEXTLIST

// ---- POUs/Alle_Rum/Gange/Gang_3_309/Visualization_4_308_1.TcVIS
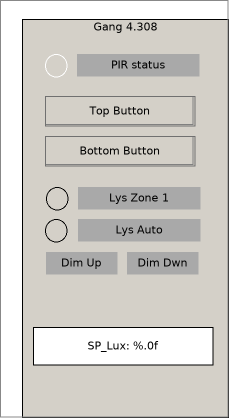
VISUALIZATION Visualization_4_308_1  // 229x418
    RoundedRectangle (22,19 207x399), "Gang 4.308"
    Rectangle (33,327 180x38), "SP_Lux: %.0f", text variable: P_Gang_4_308.arrfbLysGruppe[1].fbLightCtrl.fLuxZone1
    Button (45,96 150x30), "Top Button"
        tap P_Gang_4_308.bButtonZone1_Visu
    Button (45,136 150x30), "Bottom Button"
        tap P_Gang_4_308.bBottomButtonZone1_Visu
    Ellipse (46,187 22x23), colour toggle: P_Gang_4_308.fbLys.fbLightCtrl.bOnZone1
    Rectangle (78,187 122x22), "Lys Zone 1"
    Rectangle (46,252 71x22), "Dim Up", colour toggle: P_Gang_4_308.arrfbLysGruppe[1].fbLightCtrl.bDimUp
    Rectangle (127,252 71x22), "Dim Dwn", colour toggle: P_Gang_4_308.arrfbLysGruppe[1].fbLightCtrl.bDimDwn
    Ellipse (45,219 22x23), colour toggle: P_Gang_4_308.arrfbLysGruppe[1].fbLightCtrl.bAutoZone1
    Rectangle (78,219 122x22), "Lys Auto"
    Ellipse (45,54 22x23), colour toggle: P_Gang_4_308.arrfbLysGruppe[1].fbLightCtrl.bPIR
    Rectangle (77,54 122x22), "PIR status"
END_VISUALIZATION

// ---- POUs/Alle_Rum/Gange/Gang_4_313/Visualization_G4_313.TcVIS
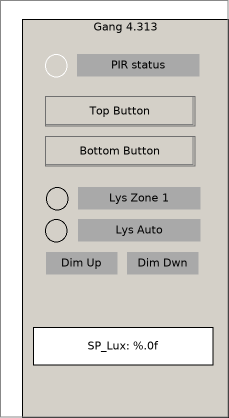
VISUALIZATION Visualization_G4_313  // 229x418
    RoundedRectangle (22,19 207x399), "Gang 4.313"
    Rectangle (33,327 180x38), "SP_Lux: %.0f", text variable: P_Gang_4_313.arrfbLysGruppe[1].fbLightCtrl.fLuxZone1
    Button (45,96 150x30), "Top Button"
        tap P_Gang_4_313.bTopButtonZone1_Visu
    Button (45,136 150x30), "Bottom Button"
        tap P_Gang_4_313.bBottomButtonZone1_Visu
    Ellipse (46,187 22x23), colour toggle: P_Gang_4_313.arrfbLysGruppe[1].fbLightCtrl.bOnZone1
    Rectangle (78,187 122x22), "Lys Zone 1"
    Rectangle (46,252 71x22), "Dim Up", colour toggle: P_Gang_4_313.arrfbLysGruppe[1].fbLightCtrl.bDimUp
    Rectangle (127,252 71x22), "Dim Dwn", colour toggle: P_Gang_4_313.arrfbLysGruppe[1].fbLightCtrl.bDimDwn
    Ellipse (45,219 22x23), colour toggle: P_Gang_4_313.arrfbLysGruppe[1].fbLightCtrl.bAutoZone1
    Rectangle (78,219 122x22), "Lys Auto"
    Ellipse (45,54 22x23), colour toggle: P_Gang_4_313.arrfbLysGruppe[1].fbLightCtrl.bPIR
    Rectangle (77,54 122x22), "PIR status"
END_VISUALIZATION

// ---- POUs/Alle_Rum/Gange/Gang_4_308/Visualization_4_308.TcVIS
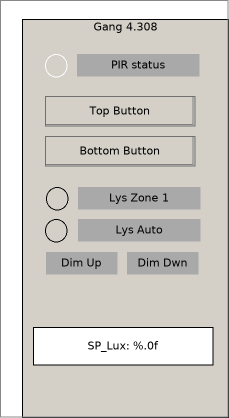
VISUALIZATION Visualization_4_308  // 229x418
    RoundedRectangle (22,19 207x399), "Gang 4.308"
    Rectangle (33,327 180x38), "SP_Lux: %.0f", text variable: P_Gang_4_308.arrfbLysGruppe[1].fbLightCtrl.fLuxZone1
    Button (45,96 150x30), "Top Button"
        tap P_Gang_4_308.bButtonZone1_Visu
    Button (45,136 150x30), "Bottom Button"
        tap P_Gang_4_308.bBottomButtonZone1_Visu
    Ellipse (46,187 22x23), colour toggle: P_Gang_4_308.fbLys.fbLightCtrl.bOnZone1
    Rectangle (78,187 122x22), "Lys Zone 1"
    Rectangle (46,252 71x22), "Dim Up", colour toggle: P_Gang_4_308.arrfbLysGruppe[1].fbLightCtrl.bDimUp
    Rectangle (127,252 71x22), "Dim Dwn", colour toggle: P_Gang_4_308.arrfbLysGruppe[1].fbLightCtrl.bDimDwn
    Ellipse (45,219 22x23), colour toggle: P_Gang_4_308.arrfbLysGruppe[1].fbLightCtrl.bAutoZone1
    Rectangle (78,219 122x22), "Lys Auto"
    Ellipse (45,54 22x23), colour toggle: P_Gang_4_308.arrfbLysGruppe[1].fbLightCtrl.bPIR
    Rectangle (77,54 122x22), "PIR status"
END_VISUALIZATION

// ---- POUs/Alle_Rum/Rum_Med_DALI_Pir/Rum_4_311/Visualization_4_311.TcVIS
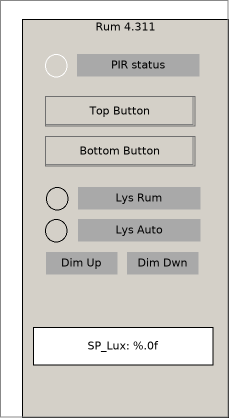
VISUALIZATION Visualization_4_311  // 229x418
    RoundedRectangle (22,19 207x399), "Rum 4.311"
    Rectangle (33,327 180x38), "SP_Lux: %.0f", text variable: P_Rum_4_311.fbLys.fbLightCtrl.fLuxZone1
    Button (45,96 150x30), "Top Button"
        tap P_Rum_4_311.bTopButtonZone1_Visu
    Button (45,136 150x30), "Bottom Button"
        tap P_Rum_4_311.bBottomButtonZone1_Visu
    Ellipse (46,187 22x23), colour toggle: P_Rum_4_311.fbLys.fbLightCtrl.bOnZone1
    Rectangle (78,187 122x22), "Lys Rum"
    Rectangle (46,252 71x22), "Dim Up", colour toggle: P_Rum_4_311.fbLys.fbLightCtrl.bDimUp
    Rectangle (127,252 71x22), "Dim Dwn", colour toggle: P_Rum_4_311.fbLys.fbLightCtrl.bDimDwn
    Ellipse (45,219 22x23), colour toggle: P_Rum_4_311.fbLys.fbLightCtrl.bAutoZone1
    Rectangle (78,219 122x22), "Lys Auto"
    Ellipse (45,54 22x23), colour toggle: P_Rum_4_311.fbLys.fbLightCtrl.bPIR
    Rectangle (77,54 122x22), "PIR status"
END_VISUALIZATION

// ---- POUs/Alle_Rum/Rum_Med_DALI_Pir/Rum_3_329/Visualization_3_329.TcVIS
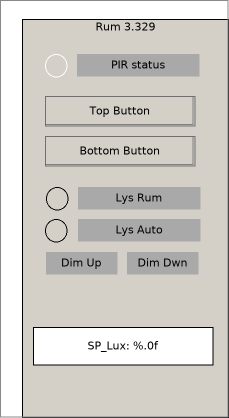
VISUALIZATION Visualization_3_329  // 229x418
    RoundedRectangle (22,19 207x399), "Rum 3.329"
    Rectangle (33,327 180x38), "SP_Lux: %.0f", text variable: P_Rum_3_329.fbLys.fbLightCtrl.fLuxZone1
    Button (45,96 150x30), "Top Button"
        tap P_Rum_3_329.bTopButtonZone1_Visu
    Button (45,136 150x30), "Bottom Button"
        tap P_Rum_3_329.bBottomButtonZone1_Visu
    Ellipse (46,187 22x23), colour toggle: P_Rum_3_329.fbLys.fbLightCtrl.bOnZone1
    Rectangle (78,187 122x22), "Lys Rum"
    Rectangle (46,252 71x22), "Dim Up", colour toggle: P_Rum_3_329.fbLys.fbLightCtrl.bDimUp
    Rectangle (127,252 71x22), "Dim Dwn", colour toggle: P_Rum_3_329.fbLys.fbLightCtrl.bDimDwn
    Ellipse (45,219 22x23), colour toggle: P_Rum_3_329.fbLys.fbLightCtrl.bAutoZone1
    Rectangle (78,219 122x22), "Lys Auto"
    Ellipse (45,54 22x23), colour toggle: P_Rum_3_329.fbLys.fbLightCtrl.bPIR
    Rectangle (77,54 122x22), "PIR status"
END_VISUALIZATION

// ---- POUs/Alle_Rum/Rum_Med_DALI_Pir/Rum_4_317/Visualization_4_316.TcVIS
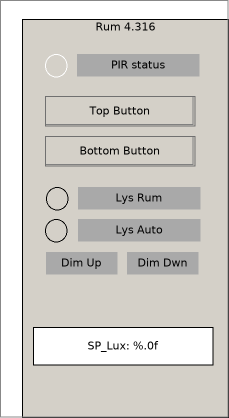
VISUALIZATION Visualization_4_316  // 229x418
    RoundedRectangle (22,19 207x399), "Rum 4.316"
    Rectangle (33,327 180x38), "SP_Lux: %.0f", text variable: P_Rum_4_316.fbLys.fbLightCtrl.fLuxZone1
    Button (45,96 150x30), "Top Button"
        tap P_Rum_4_316.bTopButtonZone1_Visu
    Button (45,136 150x30), "Bottom Button"
        tap P_Rum_4_316.bBottomButtonZone1_Visu
    Ellipse (46,187 22x23), colour toggle: P_Rum_4_316.fbLys.fbLightCtrl.bOnZone1
    Rectangle (78,187 122x22), "Lys Rum"
    Rectangle (46,252 71x22), "Dim Up", colour toggle: P_Rum_4_316.fbLys.fbLightCtrl.bDimUp
    Rectangle (127,252 71x22), "Dim Dwn", colour toggle: P_Rum_4_316.fbLys.fbLightCtrl.bDimDwn
    Ellipse (45,219 22x23), colour toggle: P_Rum_4_316.fbLys.fbLightCtrl.bAutoZone1
    Rectangle (78,219 122x22), "Lys Auto"
    Ellipse (45,54 22x23), colour toggle: P_Rum_4_316.fbLys.fbLightCtrl.bPIR
    Rectangle (77,54 122x22), "PIR status"
END_VISUALIZATION

// ---- POUs/Alle_Rum/Rum_Med_DALI_Pir/Rum_4_317/Visualization_4_317.TcVIS
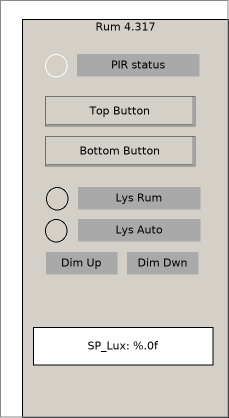
VISUALIZATION Visualization_4_317  // 229x418
    RoundedRectangle (22,19 207x399), "Rum 4.317"
    Rectangle (33,327 180x38), "SP_Lux: %.0f", text variable: P_Rum_4_317.fbLys.fbLightCtrl.fLuxZone1
    Button (45,96 150x30), "Top Button"
        tap P_Rum_4_317.bTopButtonZone1_Visu
    Button (45,136 150x30), "Bottom Button"
        tap P_Rum_4_317.bBottomButtonZone1_Visu
    Ellipse (46,187 22x23), colour toggle: P_Rum_4_317.fbLys.fbLightCtrl.bOnZone1
    Rectangle (78,187 122x22), "Lys Rum"
    Rectangle (46,252 71x22), "Dim Up", colour toggle: P_Rum_4_317.fbLys.fbLightCtrl.bDimUp
    Rectangle (127,252 71x22), "Dim Dwn", colour toggle: P_Rum_4_317.fbLys.fbLightCtrl.bDimDwn
    Ellipse (45,219 22x23), colour toggle: P_Rum_4_317.fbLys.fbLightCtrl.bAutoZone1
    Rectangle (78,219 122x22), "Lys Auto"
    Ellipse (45,54 22x23), colour toggle: P_Rum_4_317.fbLys.fbLightCtrl.bPIR
    Rectangle (77,54 122x22), "PIR status"
END_VISUALIZATION

// ---- POUs/Alle_Rum/Rum_Med_DALI_Pir/Rum_4_325_template/Visualization_4_324_1.TcVIS
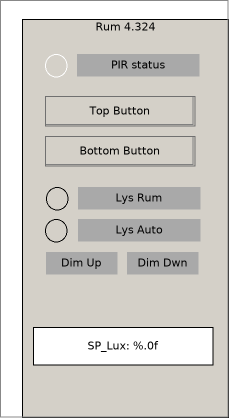
VISUALIZATION Visualization_4_324_1  // 229x418
    RoundedRectangle (22,19 207x399), "Rum 4.324"
    Rectangle (33,327 180x38), "SP_Lux: %.0f", text variable: P_Rum_4_324.fbLys.fbLightCtrl.fLuxZone1
    Button (45,96 150x30), "Top Button"
        tap P_Rum_4_324.bTopButtonZone1_Visu
    Button (45,136 150x30), "Bottom Button"
        tap P_Rum_4_324.bBottomButtonZone1_Visu
    Ellipse (46,187 22x23), colour toggle: P_Rum_4_324.fbLys.fbLightCtrl.bOnZone1
    Rectangle (78,187 122x22), "Lys Rum"
    Rectangle (46,252 71x22), "Dim Up", colour toggle: P_Rum_4_324.fbLys.fbLightCtrl.bDimUp
    Rectangle (127,252 71x22), "Dim Dwn", colour toggle: P_Rum_4_324.fbLys.fbLightCtrl.bDimDwn
    Ellipse (45,219 22x23), colour toggle: P_Rum_4_324.fbLys.fbLightCtrl.bAutoZone1
    Rectangle (78,219 122x22), "Lys Auto"
    Ellipse (45,54 22x23), colour toggle: P_Rum_4_324.fbLys.fbLightCtrl.bPIR
    Rectangle (77,54 122x22), "PIR status"
END_VISUALIZATION

// ---- POUs/DALI/DALI_Setup/VISUs/Visu_DALICommissioning/Visu_Part102SetFading.TcVIS
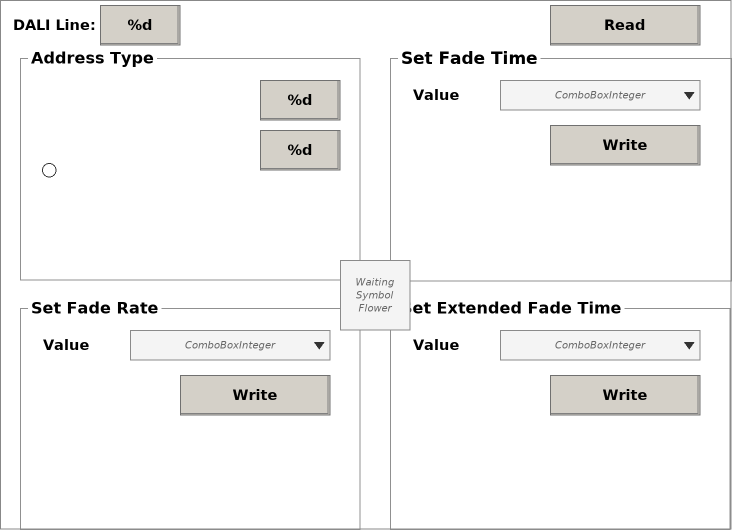
VISUALIZATION Visu_Part102SetFading  // 732x530
    GroupBox (390,50 342x231), "Set Fade Time"
        Textfield (20,30 100x30), "Value"
        ComboBoxInteger (110,30 200x30), variable: DALI_Commissioning.fbPart102SetFading.eFadeTime, text list: 'FadeTime'
        Button (160,75 150x40), "Write"
            OnMouseClick: execute { DALI_Commissioning.fbPart102SetFading.bWriteFadeTime := TRUE; }
    GroupBox (20,50 340x230), "Address Type"
        Button (240,30 80x40), "%d", text variable: DALI_Commissioning.fbPart102SetFading.nShortAddress
            OnMouseClick: write the text variable via Default, min 0, max 63, title "Insert Short Address"
        RadioButton (20,20 190x200), variable: DALI_Commissioning.fbPart102SetFading.eAddressType
            Areas[0]: Text=Short Address
            Areas[1]: Text=Group Address
            Areas[2]: Text=Broadcast
            Areas[3]: Text=Unaddressed
        Button (240,80 80x40), "%d", text variable: DALI_Commissioning.fbPart102SetFading.nGroupAddress
            OnMouseClick: write the text variable via Default, min 0, max 15, title "Insert Group Address"
    GroupBox (20,300 340x230), "Set Fade Rate"
        Textfield (20,30 100x30), "Value"
        ComboBoxInteger (110,30 200x30), variable: DALI_Commissioning.fbPart102SetFading.eFadeRate, text list: 'FadeRate'
        Button (160,75 150x40), "Write"
            OnMouseClick: execute { DALI_Commissioning.fbPart102setFading.bWriteFadeRate := TRUE; }
    GroupBox (390,300 340x230), "Set Extended Fade Time"
        Textfield (20,30 100x30), "Value"
        ComboBoxInteger (110,30 200x30), tooltip "Extended Fade Time only valid if Fade Time equals 0!", variable: DALI_Commissioning.fbPart102SetFading.eExtendedFadeTime, input disabled if: DALI_Commissioning.fbPart102SetFading.bNoFadeTime, text list: 'ExtendedFadeTime'
        Button (160,75 150x40), "Write", tooltip "Extended Fade Time only valid if Fade Time equals 0!", invisible if: DALI_Commissioning.fbPart102SetFading.bNoFadeTime, input disabled if: DALI_Commissioning.fbPart102SetFading.bNoFadeTime
            OnMouseClick: execute { DALI_Commissioning.fbPart102SetFading.bWriteExtendedFadeTime:=true; }
    Button (550,5 150x40), "Read", tooltip "Reads all Fading Parameters", invisible if: ( DALI_Commissioning.fbPart102SetFading.eAddressType >=1), input disabled if: ( DALI_Commissioning.fbPart102SetFading.eAddressType >=1)
        OnMouseClick: execute { DALI_Commissioning.fbPart102SetFading.bRead := TRUE; }
    WaitingSymbolFlower (340,260 70x70), invisible if: DALI_Commissioning.fbPart102SetFading.bHideWaitSymbol
    Group (10,5 170x40)
        Textfield (0,0 110x40), "DALI Line:"
        Button (90,0 80x40), "%d", text variable: GVL_Internal.nDALILine
            OnMouseClick: write the text variable via Default, min 1, max 10, title "Choose line"
END_VISUALIZATION

// ---- POUs/DALI/DALI_Setup/VISUs/Visu_DALICommissioning/Visu_Part103Parameters.TcVIS
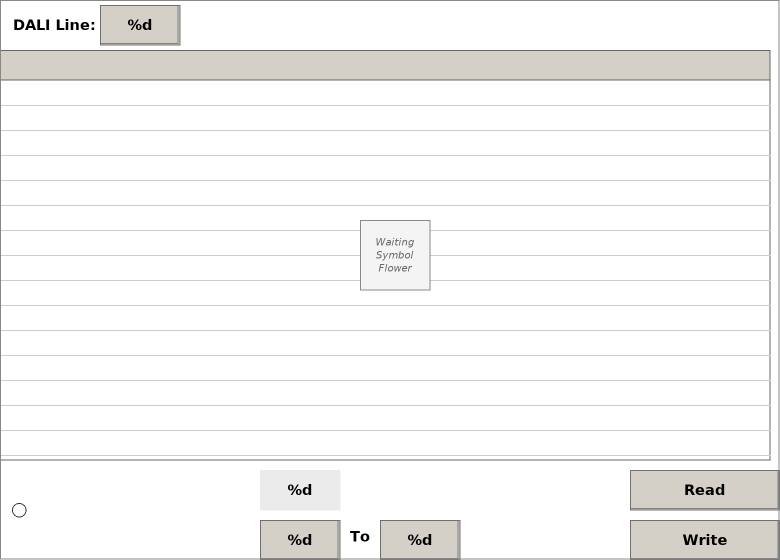
VISUALIZATION Visu_Part103Parameters  // 780x560
    Table (0,50 770x410), data array: DALI_Commissioning.fbPart103Parameters.aParameters
        p1137915858: DALI_Commissioning.fbPart103Parameters.nSelectedAddress
        p3854506369: DALI_Commissioning.fbPart103Parameters.aParameters[INDEX].nOperatingMode
        p1892666644: DALI_Commissioning.fbPart103Parameters.aParameters[INDEX].sInstanceType0
        p338671338: DALI_Commissioning.fbPart103Parameters.aParameters[INDEX].sInstanceType1
        p2170511999: DALI_Commissioning.fbPart103Parameters.aParameters[INDEX].sInstanceType2
        p3723444502: DALI_Commissioning.fbPart103Parameters.aParameters[INDEX].sInstanceType3
        p1218418051: DALI_Commissioning.fbPart103Parameters.aParameters[INDEX].sInstanceType4
        p511219082: IT0 (Generic Input)
        p1755163831: IT1 (PushButton)
        p4092479075: IT2 (Absolute Input)
        p2237128397: IT3 (Occupancy)
        p505689113: IT4 (Light Sensor)
        Columns.Column.[0].Template: OnMouseClick: write the text variable via Default, min 0, max 255, title "Insert Operating Mode 0, 128-255"
    RadioButton (10,460 230x100), variable: DALI_Commissioning.fbPart103Parameters.nAddressRange
        Areas[0]: Text=Single Short Address
        Areas[1]: Text=Short Address Range
    Textfield (260,470 80x40), "%d", text variable: DALI_Commissioning.fbPart103Parameters.nSelectedAddress
    Button (260,520 80x40), "%d", text variable: DALI_Commissioning.fbPart103Parameters.nStartAddress
        OnMouseClick: write the text variable via Default, min 0, max 63, title "Insert Short Address"
    Button (380,520 80x40), "%d", text variable: DALI_Commissioning.fbPart103Parameters.nEndAddress
        OnMouseClick: write the text variable via Default, min 0, max 63, title "Insert Short Address"
    Button (630,470 150x40), "Read"
        OnMouseClick: execute { DALI_Commissioning.fbPart103Parameters.bRead := true; }
    Button (630,520 150x40), "Write"
        OnMouseClick: execute { DALI_Commissioning.fbPart103Parameters.bWrite := true; }
    Textfield (335,521 50x31), "To"
    WaitingSymbolFlower (360,220 70x70), invisible if: DALI_Commissioning.fbPart103Parameters.bHideWaitSymbol
    Group (10,5 170x40)
        Textfield (0,0 110x40), "DALI Line:"
        Button (90,0 80x40), "%d", text variable: GVL_Internal.nDALILine
            OnMouseClick: write the text variable via Default, min 1, max 10, title "Choose line"
END_VISUALIZATION

// ---- POUs/DALI/DALI_Setup/VISUs/Visu_DALICommissioning/Visu_Part202Parameters.TcVIS
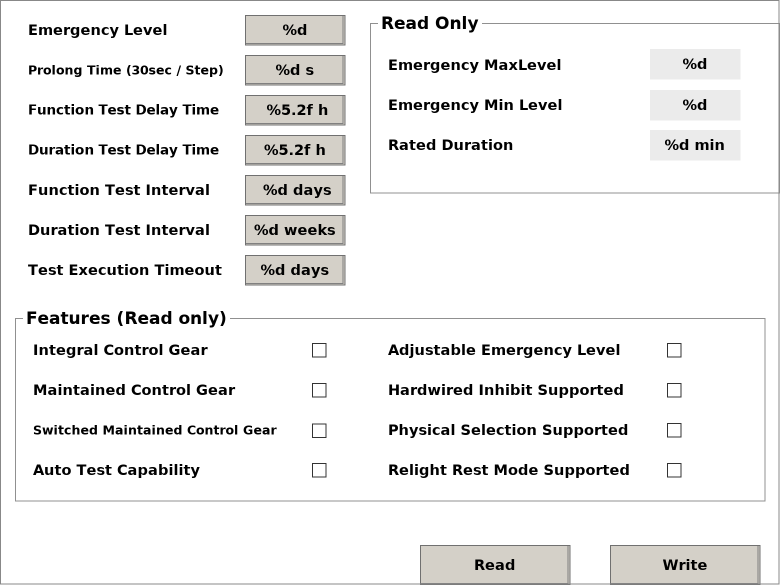
VISUALIZATION Visu_Part202Parameters  // 780x585
    Button (610,545 150x40), "Write"
        OnMouseClick: execute { DALI_Commissioning.fbPart202Emergency.bWrite:=TRUE; }
    GroupBox (15,310 750x191), "Features (Read only)"
        Textfield (15,25 250x30), "Integral Control Gear"
        Textfield (15,65 250x30), "Maintained Control Gear"
        Checkbox (295,105 30x31), variable: DALI_Commissioning.fbPart202Emergency.bSwitchtedMaintainedControlGear, input disabled if: TRUE
        Checkbox (295,25 30x30), variable: DALI_Commissioning.fbPart202Emergency.bIntegralControlGear, input disabled if: TRUE
        Checkbox (295,65 30x30), variable: DALI_Commissioning.fbPart202Emergency.bMaintainedControlGear, input disabled if: TRUE
        Textfield (370,105 250x30), "Physical Selection Supported"
        Textfield (15,145 250x30), "Auto Test Capability"
        Textfield (370,25 250x30), "Adjustable Emergency Level"
        Textfield (370,65 250x30), "Hardwired Inhibit Supported"
        Textfield (370,145 250x30), "Relight Rest Mode Supported"
        Checkbox (650,25 30x30), variable: DALI_Commissioning.fbPart202Emergency.bAdjustableEmergencyLevel, input disabled if: TRUE
        Checkbox (650,65 30x30), variable: DALI_Commissioning.fbPart202Emergency.bHardwiredInhibitSupported, input disabled if: TRUE
        Checkbox (650,105 30x30), variable: DALI_Commissioning.fbPart202Emergency.bPhysicalSelectionSupported, input disabled if: TRUE
        Checkbox (650,145 30x30), variable: DALI_Commissioning.fbPart202Emergency.bRelightinRestModeSupported, input disabled if: TRUE
        Textfield (15,105 250x30), "Switched Maintained Control Gear"
        Checkbox (295,145 30x30), variable: DALI_Commissioning.fbPart202Emergency.bAutoTestCapability, input disabled if: TRUE
    Textfield (25,15 200x30), "Emergency Level"
    Textfield (25,95 200x30), "Function Test Delay Time"
    Textfield (25,135 200x30), "Duration Test Delay Time"
    Button (245,15 100x30), "%d", text variable: DALI_Commissioning.fbPart202Emergency.nEmergencyLevel
        OnMouseClick: write the text variable via Default, min 0, max 255, title "Emergency Level"
    Button (245,95 100x30), "%5.2f h", text variable: DALI_Commissioning.fbPart205Incandescent.fLoadRating
        OnMouseClick: write the text variable via Default, min 0, max 16384, title "Function Test Delay Time"
    Button (245,135 100x30), "%5.2f h", text variable: DALI_Commissioning.fbPart202Emergency.fDurationTestDelayTimeVisu
        OnMouseClick: write the text variable via Default, min 0, max 16384, title "Duration Test Delay Time"
    Textfield (25,55 200x30), "Prolong Time (30sec / Step)"
    Button (245,55 100x30), "%d s", text variable: DALI_Commissioning.fbPart202Emergency.nProlongTime
        OnMouseClick: write the text variable via Default, min 0, max 255, title "Prolong Time"
    Textfield (25,255 200x30), "Test Execution Timeout"
    Button (245,255 100x30), "%d days", text variable: DALI_Commissioning.fbPart202Emergency.nTestExecutionTimeout
        OnMouseClick: write the text variable via Default, min 0, max 255, title "Test Execution Timeout"
    GroupBox (370,15 410x178), "Read Only"
        Textfield (15,115 220x30), "Rated Duration"
        Textfield (15,75 220x30), "Emergency Min Level"
        Textfield (15,35 220x30), "Emergency MaxLevel"
        Textfield (280,34 90x30), "%d", text variable: DALI_Commissioning.fbPart202Emergency.nEmergencyMaxLevel
        Textfield (280,75 90x30), "%d", text variable: DALI_Commissioning.fbPart202Emergency.nEmergencyMinLevel
        Textfield (280,115 90x30), "%d min", text variable: DALI_Commissioning.fbPart202Emergency.nRatedDuration
    Textfield (25,175 200x30), "Function Test Interval"
    Textfield (25,215 200x30), "Duration Test Interval"
    Button (245,175 100x30), "%d days", text variable: DALI_Commissioning.fbPart202Emergency.nFunctionTestInterval
        OnMouseClick: write the text variable via Default, min 0, max 255, title "Function Test Delay Time"
    Button (245,215 100x30), "%d weeks", text variable: DALI_Commissioning.fbPart202Emergency.nDurationTestInterval
        OnMouseClick: write the text variable via Default, min 0, max 255, title "Duration Test Delay Time"
    Button (420,545 150x40), "Read"
        OnMouseClick: execute { DALI_Commissioning.fbPart202Emergency.bReadParameter:=TRUE; }
END_VISUALIZATION

// ---- POUs/DALI/DALI_Setup/VISUs/Visu_DALICommissioning/Visu_Part202Status.TcVIS
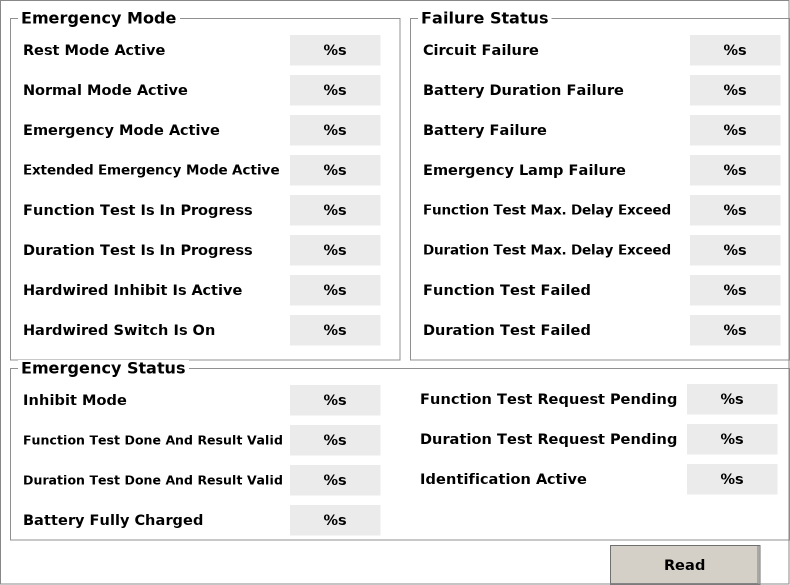
VISUALIZATION Visu_Part202Status  // 790x585
    Button (610,545 150x40), "Read"
        OnMouseClick: execute { DALI_Commissioning.fbPart202Emergency.bReadState:=TRUE; }
    GroupBox (10,10 390x350), "Emergency Mode"
        Textfield (10,145 260x30), "Extended Emergency Mode Active"
        Textfield (280,185 90x30), "%s", text variable: DALI_Commissioning.fbPart202Emergency.sFunctionTest
        Textfield (280,145 90x30), "%s", text variable: DALI_Commissioning.fbPart202Emergency.sExtendedEmergency
        Textfield (280,105 90x30), "%s", text variable: DALI_Commissioning.fbPart202Emergency.sEmergencyMode
        Textfield (280,65 90x30), "%s", text variable: DALI_Commissioning.fbPart202Emergency.sNormalMode
        Textfield (280,25 90x30), "%s", text variable: DALI_Commissioning.fbPart202Emergency.sRestMode
        Textfield (10,25 260x30), "Rest Mode Active"
        Textfield (10,65 260x30), "Normal Mode Active"
        Textfield (10,105 260x30), "Emergency Mode Active"
        Textfield (10,185 260x30), "Function Test Is In Progress"
        Textfield (10,225 260x30), "Duration Test Is In Progress"
        Textfield (10,265 260x30), "Hardwired Inhibit Is Active"
        Textfield (10,305 260x30), "Hardwired Switch Is On"
        Textfield (280,265 90x30), "%s", text variable: DALI_Commissioning.fbPart202Emergency.sHardwiredInhibit
        Textfield (280,305 90x30), "%s", text variable: DALI_Commissioning.fbPart202Emergency.sHardwiredSwitch
        Textfield (280,225 90x30), "%s", text variable: DALI_Commissioning.fbPart202Emergency.sDurationTest
    GroupBox (410,10 380x350), "Failure Status"
        Textfield (10,145 260x30), "Emergency Lamp Failure"
        Textfield (280,185 90x30), "%s", text variable: DALI_Commissioning.fbPart202Emergency.sFunctionTestExceed
        Textfield (280,145 90x30), "%s", text variable: DALI_Commissioning.fbPart202Emergency.sEmergencyLampFailure
        Textfield (280,105 90x30), "%s", text variable: DALI_Commissioning.fbPart202Emergency.sBatteryFailure
        Textfield (280,65 90x30), "%s", text variable: DALI_Commissioning.fbPart202Emergency.sBatteryDurationFailure
        Textfield (280,25 90x30), "%s", text variable: DALI_Commissioning.fbPart202Emergency.sCircuitFailure
        Textfield (10,25 260x30), "Circuit Failure"
        Textfield (10,65 260x30), "Battery Duration Failure"
        Textfield (10,105 260x30), "Battery Failure"
        Textfield (10,185 260x30), "Function Test Max. Delay Exceed"
        Textfield (10,225 260x30), "Duration Test Max. Delay Exceed"
        Textfield (10,265 260x30), "Function Test Failed"
        Textfield (10,305 260x30), "Duration Test Failed"
        Textfield (280,265 90x30), "%s", text variable: DALI_Commissioning.fbPart202Emergency.sFunctionTestFailed
        Textfield (280,305 90x30), "%s", text variable: DALI_Commissioning.fbPart202Emergency.sDurationTestFailed
        Textfield (280,225 90x30), "%s", text variable: DALI_Commissioning.fbPart202Emergency.sDurationTestExceed
    GroupBox (10,360 780x180), "Emergency Status"
        Textfield (10,145 260x30), "Battery Fully Charged"
        Textfield (677,24 90x30), "%s", text variable: DALI_Commissioning.fbPart202Emergency.sFunctionTestRequestPending
        Textfield (10,25 260x30), "Inhibit Mode"
        Textfield (10,65 260x30), "Function Test Done And Result Valid"
        Textfield (407,24 260x30), "Function Test Request Pending"
        Textfield (407,64 260x30), "Duration Test Request Pending"
        Textfield (407,104 260x30), "Identification Active"
        Textfield (677,104 90x30), "%s", text variable: DALI_Commissioning.fbPart202Emergency.sIdentificationActive
        Textfield (677,64 90x30), "%s", text variable: DALI_Commissioning.fbPart202Emergency.sDurationTestRequestPending
        Textfield (280,25 90x30), "%s", text variable: DALI_Commissioning.fbPart202Emergency.sInhibitMode
        Textfield (280,65 90x30), "%s", text variable: DALI_Commissioning.fbPart202Emergency.sFunctionTestDoneValid
        Textfield (280,145 90x30), "%s", text variable: DALI_Commissioning.fbPart202Emergency.sBatteryFullCharged
        Textfield (10,105 260x30), "Duration Test Done And Result Valid"
        Textfield (280,105 90x30), "%s", text variable: DALI_Commissioning.fbPart202Emergency.sDurationTestDoneValid
END_VISUALIZATION

// ---- POUs/DALI/DALI_Setup/VISUs/Visu_DALICommissioning/Visu_Part207.TcVIS
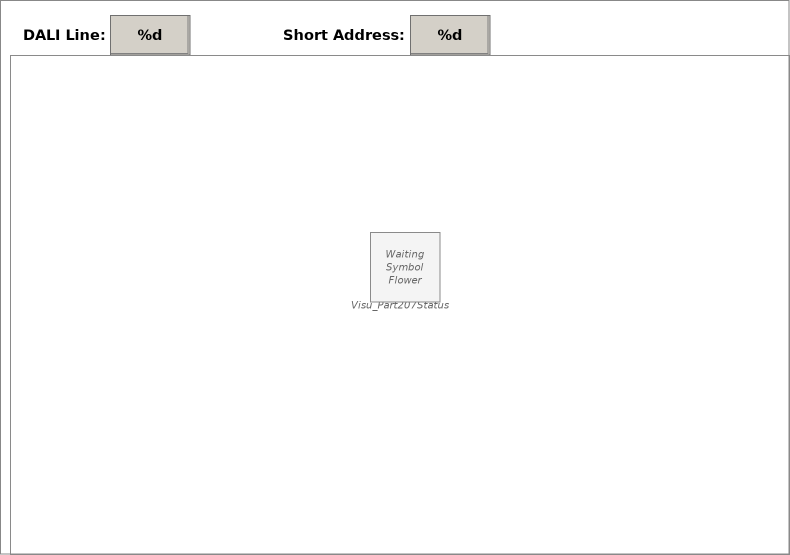
VISUALIZATION Visu_Part207  // 790x555
    Group (280,15 210x40)
        Textfield (0,0 130x40), "Short Address:"
        Button (130,0 80x40), "%d", text variable: DALI_Commissioning.fbPart207LED.nAddress
            OnMouseClick: write the text variable via Default, min 0, max 63, title "Insert Short Address"
    Group (20,15 170x40)
        Textfield (0,0 110x40), "DALI Line:"
        Button (90,0 80x40), "%d", text variable: GVL_Internal.nDALILine
            OnMouseClick: write the text variable via Default, min 1, max 10, title "Choose line"
    TabControl (10,55 780x500)
        shows Visu_Part207Status()
        shows Visu_Part207Parameters()
        shows Test()
        [0]: TabTitle=Status LED
        [1]: TabTitle=Parameters LED
        [2]: TabTitle=Paremeters LED
    WaitingSymbolFlower (370,232 70x70), invisible if: DALI_Commissioning.fbPart207LED.bHideWaitSymbol
END_VISUALIZATION
